C03636=1093.569,93.701,438.631,175.911,17.516,152.546
C03637=1093.575,93.950,438.614,175.913,17.517,152.546
C03638=1093.581,94.199,438.595,175.915,17.518,152.546
C03639=1093.586,94.448,438.577,175.918,17.519,152.546
C03640=1093.592,94.697,438.559,175.920,17.520,152.545
C03641=1093.598,94.947,438.541,175.923,17.521,152.545
C03642=1093.603,95.196,438.524,175.925,17.522,152.545
C03643=1093.609,95.472,438.503,175.927,17.523,152.545
C03644=1093.616,95.748,438.484,175.930,17.524,152.544
C03645=1093.622,96.023,438.464,175.933,17.525,152.544
C03646=1093.628,96.299,438.443,175.935,17.526,152.544
C03647=1093.634,96.548,438.425,175.938,17.528,152.544
C03648=1093.639,96.797,438.408,175.940,17.529,152.543
C03649=1093.645,97.048,438.389,175.942,17.530,152.543
C03650=1093.651,97.296,438.371,175.944,17.531,152.543
C03651=1093.657,97.546,438.353,175.947,17.532,152.543
C03652=1093.662,97.795,438.336,175.950,17.533,152.542
C03653=1093.668,98.045,438.317,175.952,17.534,152.542
C03654=1093.673,98.293,438.299,175.954,17.535,152.542
C03655=1093.680,98.543,438.281,175.956,17.535,152.542
C03656=1093.684,98.792,438.263,175.959,17.537,152.541
C03657=1093.691,99.041,438.244,175.961,17.537,152.541
C03658=1093.696,99.290,438.227,175.964,17.538,152.541
C03659=1093.702,99.540,438.209,175.966,17.540,152.541
C03660=1093.707,99.789,438.190,175.968,17.540,152.540
C03661=1093.714,100.039,438.172,175.971,17.541,152.540
C03662=1093.719,100.288,438.154,175.973,17.542,152.540
C03663=1093.725,100.537,438.135,175.976,17.543,152.540
C03664=1093.730,100.786,438.117,175.978,17.545,152.539
C03665=1093.736,101.036,438.099,175.980,17.545,152.539
C03666=1093.742,101.285,438.081,175.983,17.546,152.539
C03667=1093.748,101.534,438.063,175.985,17.547,152.538
C03668=1093.753,101.783,438.044,175.988,17.548,152.538
C03669=1093.759,102.033,438.026,175.990,17.549,152.538
C03670=1093.764,102.282,438.007,175.992,17.550,152.538
C03671=1093.770,102.531,437.989,175.995,17.551,152.537
C03672=1093.775,102.781,437.971,175.998,17.552,152.537
C03673=1093.781,103.030,437.952,176.000,17.553,152.537
C03674=1093.786,103.279,437.934,176.002,17.554,152.537
C03675=1093.792,103.528,437.915,176.004,17.555,152.536
C03676=1093.797,103.778,437.897,176.007,17.556,152.536
C03677=1093.804,104.027,437.879,176.010,17.557,152.536
C03678=1093.808,104.276,437.860,176.012,17.558,152.536
C03679=1093.815,104.525,437.842,176.014,17.559,152.535
C03680=1093.820,104.775,437.824,176.016,17.559,152.535
C03681=1093.826,105.024,437.805,176.019,17.560,152.535
C03682=1093.831,105.273,437.787,176.022,17.562,152.534
C03683=1093.837,105.522,437.768,176.024,17.562,152.534
C03684=1093.842,105.771,437.749,176.027,17.563,152.534
C03685=1093.848,106.021,437.731,176.029,17.565,152.534
C03686=1093.854,106.269,437.712,176.031,17.565,152.533
C03687=1093.859,106.519,437.694,176.034,17.566,152.533
C03688=1093.865,106.769,437.675,176.036,17.567,152.533
C03689=1093.870,107.017,437.656,176.039,17.568,152.532
C03690=1093.877,107.267,437.638,176.041,17.569,152.532
C03691=1093.882,107.516,437.620,176.043,17.570,152.532
C03692=1093.887,107.766,437.601,176.046,17.571,152.532
C03693=1093.893,108.015,437.582,176.049,17.572,152.531
C03694=1093.899,108.264,437.564,176.051,17.573,152.531
C03695=1093.905,108.513,437.546,176.054,17.573,152.531
C03696=1093.910,108.762,437.527,176.056,17.574,152.530
C03697=1093.915,109.012,437.508,176.058,17.575,152.530
C03698=1093.922,109.261,437.490,176.061,17.576,152.530
C03699=1093.927,109.510,437.471,176.063,17.577,152.530
C03700=1093.933,109.759,437.452,176.066,17.578,152.529
C03701=1093.939,110.009,437.433,176.069,17.579,152.529
C03702=1093.944,110.258,437.415,176.071,17.580,152.529
C03703=1093.950,110.507,437.396,176.073,17.581,152.528
C03704=1093.956,110.757,437.377,176.075,17.581,152.528
C03705=1093.962,111.005,437.358,176.078,17.582,152.528
C03706=1093.967,111.255,437.340,176.081,17.583,152.528
C03707=1093.973,111.531,437.319,176.084,17.584,152.527
C03708=1093.979,111.806,437.298,176.087,17.585,152.527
C03709=1093.985,112.082,437.277,176.089,17.586,152.527
C03710=1093.992,112.359,437.256,176.092,17.587,152.526
C03711=1093.997,112.607,437.238,176.094,17.588,152.526
C03712=1094.003,112.856,437.219,176.097,17.589,152.526
C03713=1094.009,113.106,437.199,176.099,17.589,152.525
C03714=1094.014,113.355,437.181,176.102,17.590,152.525
C03715=1094.020,113.604,437.163,176.105,17.592,152.525
C03716=1094.026,113.854,437.143,176.107,17.592,152.524
C03717=1094.031,114.103,437.124,176.109,17.593,152.524
C03718=1094.036,114.352,437.105,176.112,17.594,152.524
C03719=1094.043,114.601,437.087,176.114,17.595,152.524
C03720=1094.049,114.850,437.067,176.117,17.595,152.523
C03721=1094.054,115.099,437.048,176.120,17.597,152.523
C03722=1094.059,115.349,437.029,176.122,17.597,152.523
C03723=1094.065,115.598,437.010,176.124,17.598,152.522
C03724=1094.070,115.847,436.991,176.127,17.599,152.522
C03725=1094.076,116.096,436.972,176.129,17.600,152.522
C03726=1094.081,116.346,436.953,176.132,17.601,152.521
C03727=1094.086,116.595,436.934,176.134,17.602,152.521
C03728=1094.092,116.844,436.915,176.137,17.602,152.521
C03729=1094.098,117.094,436.896,176.140,17.604,152.520
C03730=1094.103,117.343,436.877,176.142,17.604,152.520
C03731=1094.108,117.592,436.858,176.145,17.605,152.520
C03732=1094.114,117.842,436.839,176.147,17.606,152.520
C03733=1094.119,118.090,436.820,176.149,17.607,152.519
C03734=1094.126,118.339,436.801,176.152,17.607,152.519
C03735=1094.132,118.588,436.781,176.155,17.609,152.519
C03736=1094.137,118.838,436.762,176.157,17.609,152.518
C03737=1094.142,119.086,436.743,176.160,17.610,152.518
C03738=1094.148,119.336,436.724,176.163,17.611,152.518
C03739=1094.154,119.585,436.705,176.165,17.611,152.517
C03740=1094.159,119.835,436.685,176.167,17.613,152.517
C03741=1094.165,120.083,436.666,176.170,17.614,152.517
C03742=1094.170,120.333,436.647,176.172,17.614,152.516
C03743=1094.176,120.582,436.628,176.175,17.615,152.516
C03744=1094.182,120.832,436.609,176.178,17.616,152.516
C03745=1094.187,121.080,436.590,176.181,17.617,152.515
C03746=1094.193,121.329,436.570,176.183,17.617,152.515
C03747=1094.198,121.579,436.551,176.186,17.618,152.515
C03748=1094.204,121.828,436.531,176.188,17.620,152.515
C03749=1094.210,122.078,436.512,176.191,17.620,152.514
C03750=1094.215,122.326,436.493,176.193,17.621,152.514
C03751=1094.220,122.575,436.473,176.196,17.622,152.513
C03752=1094.226,122.825,436.453,176.198,17.622,152.513
C03753=1094.231,123.074,436.434,176.201,17.623,152.513
C03754=1094.237,123.324,436.415,176.204,17.624,152.512
C03755=1094.242,123.572,436.396,176.206,17.624,152.512
C03756=1094.248,123.821,436.376,176.209,17.626,152.512
C03757=1094.254,124.071,436.357,176.212,17.626,152.511
C03758=1094.260,124.320,436.338,176.214,17.627,152.511
C03759=1094.266,124.569,436.318,176.217,17.628,152.511
C03760=1094.271,124.818,436.298,176.220,17.628,152.510
C03761=1094.277,125.068,436.279,176.222,17.629,152.510
C03762=1094.282,125.316,436.260,176.225,17.630,152.510
C03763=1094.288,125.565,436.240,176.227,17.631,152.509
C03764=1094.294,125.815,436.221,176.229,17.631,152.509
C03765=1094.299,126.064,436.202,176.232,17.632,152.509
C03766=1094.305,126.313,436.181,176.235,17.633,152.508
C03767=1094.310,126.563,436.162,176.238,17.634,152.508
C03768=1094.316,126.812,436.142,176.240,17.634,152.508
C03769=1094.322,127.061,436.123,176.243,17.635,152.507
C03770=1094.328,127.310,436.104,176.246,17.636,152.507
C03771=1094.334,127.586,436.082,176.249,17.637,152.506
C03772=1094.340,127.862,436.060,176.252,17.638,152.506
C03773=1094.347,128.138,436.039,176.255,17.639,152.506
C03774=1094.353,128.413,436.017,176.258,17.639,152.505
C03775=1094.358,128.663,435.997,176.260,17.639,152.505
C03776=1094.364,128.912,435.977,176.263,17.641,152.505
C03777=1094.370,129.161,435.958,176.266,17.641,152.504
C03778=1094.376,129.410,435.938,176.268,17.642,152.504
C03779=1094.382,129.659,435.919,176.271,17.642,152.503
C03780=1094.388,129.908,435.899,176.274,17.643,152.503
C03781=1094.393,130.158,435.879,176.276,17.644,152.503
C03782=1094.398,130.407,435.859,176.279,17.644,152.502
C03783=1094.404,130.656,435.840,176.282,17.645,152.502
C03784=1094.410,130.905,435.820,176.284,17.646,152.502
C03785=1094.416,131.154,435.800,176.287,17.646,152.501
C03786=1094.422,131.403,435.780,176.290,17.647,152.501
C03787=1094.427,131.653,435.761,176.293,17.648,152.500
C03788=1094.433,131.902,435.741,176.294,17.649,152.500
C03789=1094.439,132.151,435.721,176.297,17.649,152.500
C03790=1094.444,132.400,435.701,176.300,17.650,152.499
C03791=1094.450,132.649,435.681,176.303,17.650,152.499
C03792=1094.455,132.898,435.662,176.305,17.651,152.499
C03793=1094.461,133.147,435.642,176.308,17.652,152.498
C03794=1094.466,133.396,435.621,176.311,17.653,152.498
C03795=1094.472,133.645,435.602,176.313,17.653,152.498
C03796=1094.477,133.894,435.582,176.316,17.654,152.497
C03797=1094.483,134.144,435.562,176.319,17.655,152.497
C03798=1094.489,134.393,435.542,176.322,17.656,152.496
C03799=1094.494,134.642,435.522,176.324,17.656,152.496
C03800=1094.500,134.891,435.502,176.327,17.657,152.496
C03801=1094.505,135.140,435.482,176.330,17.658,152.495
C03802=1094.511,135.389,435.462,176.332,17.658,152.495
C03803=1094.517,135.638,435.442,176.335,17.659,152.495
C03804=1094.522,135.888,435.422,176.338,17.659,152.494
C03805=1094.528,136.137,435.402,176.341,17.661,152.494
C03806=1094.534,136.386,435.381,176.343,17.661,152.493
C03807=1094.540,136.635,435.362,176.346,17.661,152.493
C03808=1094.545,136.885,435.342,176.349,17.662,152.493
C03809=1094.551,137.134,435.322,176.352,17.663,152.492
C03810=1094.557,137.383,435.302,176.354,17.663,152.492
C03811=1094.562,137.632,435.281,176.357,17.664,152.492
C03812=1094.568,137.880,435.261,176.360,17.665,152.491
C03813=1094.573,138.130,435.241,176.362,17.665,152.491
C03814=1094.579,138.379,435.221,176.365,17.666,152.490
C03815=1094.584,138.628,435.201,176.368,17.667,152.490
C03816=1094.590,138.877,435.181,176.371,17.667,152.490
C03817=1094.595,139.126,435.160,176.373,17.668,152.489
C03818=1094.601,139.375,435.140,176.376,17.668,152.489
C03819=1094.606,139.625,435.121,176.379,17.669,152.488
C03820=1094.613,139.874,435.100,176.382,17.670,152.488
C03821=1094.618,140.123,435.080,176.384,17.670,152.488
C03822=1094.624,140.372,435.060,176.387,17.671,152.487
C03823=1094.629,140.621,435.039,176.390,17.672,152.487
C03824=1094.635,140.870,435.019,176.393,17.673,152.486
C03825=1094.641,141.119,434.999,176.395,17.673,152.486
C03826=1094.646,141.368,434.978,176.398,17.674,152.486
C03827=1094.652,141.617,434.958,176.401,17.674,152.485
C03828=1094.657,141.866,434.938,176.404,17.675,152.485
C03829=1094.662,142.115,434.917,176.406,17.675,152.484
C03830=1094.669,142.365,434.897,176.409,17.676,152.484
C03831=1094.674,142.614,434.876,176.412,17.677,152.484
C03832=1094.679,142.863,434.856,176.415,17.677,152.483
C03833=1094.685,143.112,434.836,176.418,17.678,152.483
C03834=1094.691,143.361,434.815,176.420,17.679,152.482
C03835=1094.697,143.637,434.793,176.424,17.679,152.482
C03836=1094.703,143.913,434.770,176.427,17.680,152.482
C03837=1094.709,144.189,434.747,176.430,17.681,152.481
C03838=1094.715,144.464,434.725,176.432,17.681,152.481
C03839=1094.721,144.713,434.705,176.435,17.682,152.480
C03840=1094.726,144.962,434.684,176.438,17.683,152.480
C03841=1094.732,145.212,434.663,176.441,17.683,152.479
C03842=1094.739,145.460,434.643,176.444,17.684,152.479
C03843=1094.744,145.709,434.622,176.447,17.684,152.479
C03844=1094.749,145.958,434.601,176.450,17.685,152.478
C03845=1094.754,146.208,434.581,176.453,17.685,152.478
C03846=1094.761,146.457,434.561,176.455,17.686,152.477
C03847=1094.766,146.706,434.540,176.458,17.686,152.477
C03848=1094.771,146.955,434.519,176.461,17.687,152.476
C03849=1094.778,147.203,434.499,176.464,17.688,152.476
C03850=1094.784,147.453,434.478,176.467,17.689,152.476
C03851=1094.789,147.702,434.457,176.469,17.689,152.475
C03852=1094.794,147.952,434.437,176.472,17.689,152.475
C03853=1094.800,148.200,434.417,176.475,17.690,152.474
C03854=1094.806,148.449,434.396,176.478,17.690,152.474
C03855=1094.812,148.699,434.375,176.481,17.691,152.473
C03856=1094.817,148.948,434.354,176.484,17.691,152.473
C03857=1094.822,149.197,434.334,176.487,17.692,152.473
C03858=1094.828,149.445,434.312,176.490,17.693,152.472
C03859=1094.834,149.695,434.292,176.493,17.694,152.472
C03860=1094.839,149.944,434.271,176.495,17.694,152.471
C03861=1094.845,150.193,434.250,176.498,17.694,152.471
C03862=1094.850,150.442,434.230,176.501,17.695,152.471
C03863=1094.856,150.692,434.209,176.504,17.695,152.470
C03864=1094.862,150.940,434.187,176.506,17.696,152.470
C03865=1094.867,151.189,434.167,176.509,17.696,152.469
C03866=1094.872,151.438,434.146,176.512,17.697,152.469
C03867=1094.878,151.687,434.125,176.515,17.698,152.468
C03868=1094.884,151.936,434.105,176.518,17.699,152.468
C03869=1094.890,152.185,434.084,176.520,17.698,152.467
C03870=1094.896,152.435,434.062,176.523,17.699,152.467
C03871=1094.901,152.684,434.042,176.526,17.700,152.467
C03872=1094.907,152.932,434.021,176.529,17.701,152.466
C03873=1094.912,153.181,434.000,176.532,17.701,152.466
C03874=1094.918,153.431,433.979,176.535,17.701,152.465
C03875=1094.923,153.680,433.958,176.538,17.702,152.465
C03876=1094.929,153.929,433.937,176.541,17.702,152.464
C03877=1094.935,154.178,433.916,176.544,17.703,152.464
C03878=1094.940,154.427,433.895,176.547,17.704,152.463
C03879=1094.946,154.676,433.874,176.549,17.704,152.463
C03880=1094.951,154.925,433.853,176.552,17.704,152.463
C03881=1094.957,155.174,433.832,176.555,17.705,152.462
C03882=1094.962,155.423,433.811,176.559,17.705,152.462
C03883=1094.968,155.672,433.790,176.561,17.706,152.461
C03884=1094.974,155.921,433.769,176.564,17.706,152.461
C03885=1094.979,156.170,433.748,176.567,17.707,152.460
C03886=1094.985,156.420,433.727,176.570,17.707,152.460
C03887=1094.991,156.668,433.706,176.573,17.708,152.460
C03888=1094.997,156.917,433.684,176.576,17.709,152.459
C03889=1095.002,157.167,433.663,176.578,17.709,152.459
C03890=1095.008,157.415,433.642,176.581,17.709,152.458
C03891=1095.013,157.665,433.621,176.584,17.710,152.458
C03892=1095.018,157.914,433.599,176.587,17.711,152.457
C03893=1095.024,158.162,433.578,176.591,17.711,152.457
C03894=1095.030,158.412,433.557,176.594,17.712,152.456
C03895=1095.035,158.661,433.536,176.596,17.712,152.456
C03896=1095.041,158.910,433.514,176.599,17.712,152.455
C03897=1095.047,159.159,433.494,176.602,17.713,152.455
C03898=1095.052,159.407,433.472,176.605,17.714,152.455
C03899=1095.058,159.683,433.448,176.608,17.714,152.454
C03900=1095.065,159.958,433.425,176.611,17.714,152.453
C03901=1095.071,160.234,433.401,176.614,17.715,152.453
C03902=1095.077,160.509,433.378,176.618,17.715,152.453
C03903=1095.083,160.759,433.357,176.621,17.716,152.452
C03904=1095.088,161.008,433.335,176.624,17.716,152.452
C03905=1095.094,161.256,433.314,176.627,17.717,152.451
C03906=1095.099,161.506,433.292,176.630,17.717,152.451
C03907=1095.105,161.754,433.271,176.632,17.718,152.450
C03908=1095.111,162.004,433.250,176.635,17.718,152.450
C03909=1095.116,162.253,433.228,176.639,17.719,152.449
C03910=1095.121,162.501,433.207,176.642,17.719,152.449
C03911=1095.127,162.751,433.185,176.645,17.720,152.448
C03912=1095.132,162.999,433.163,176.648,17.720,152.448
C03913=1095.138,163.249,433.142,176.651,17.721,152.447
C03914=1095.143,163.498,433.120,176.653,17.721,152.447
C03915=1095.149,163.747,433.099,176.656,17.722,152.446
C03916=1095.155,163.996,433.077,176.659,17.722,152.446
C03917=1095.159,164.245,433.055,176.662,17.723,152.446
C03918=1095.166,164.494,433.034,176.665,17.723,152.445
C03919=1095.170,164.743,433.012,176.668,17.724,152.445
C03920=1095.176,164.992,432.991,176.671,17.724,152.444
C03921=1095.181,165.241,432.969,176.674,17.725,152.444
C03922=1095.187,165.490,432.948,176.677,17.725,152.443
C03923=1095.193,165.739,432.926,176.680,17.726,152.443
C03924=1095.198,165.988,432.904,176.683,17.726,152.442
C03925=1095.204,166.237,432.883,176.686,17.727,152.442
C03926=1095.209,166.486,432.861,176.689,17.728,152.441
C03927=1095.215,166.735,432.839,176.691,17.728,152.441
C03928=1095.220,166.984,432.817,176.695,17.728,152.440
C03929=1095.226,167.233,432.796,176.698,17.729,152.440
C03930=1095.231,167.482,432.774,176.701,17.729,152.439
C03931=1095.237,167.731,432.752,176.704,17.730,152.439
C03932=1095.242,167.980,432.730,176.707,17.730,152.439
C03933=1095.248,168.229,432.709,176.710,17.731,152.438
C03934=1095.253,168.478,432.687,176.713,17.731,152.438
C03935=1095.259,168.727,432.665,176.716,17.731,152.437
C03936=1095.264,168.975,432.643,176.719,17.732,152.437
C03937=1095.270,169.224,432.621,176.722,17.732,152.436
C03938=1095.276,169.474,432.599,176.725,17.733,152.436
C03939=1095.281,169.723,432.578,176.728,17.733,152.435
C03940=1095.287,169.972,432.555,176.731,17.734,152.435
C03941=1095.292,170.221,432.534,176.734,17.734,152.434
C03942=1095.297,170.470,432.512,176.737,17.734,152.434
C03943=1095.303,170.719,432.491,176.740,17.735,152.433
C03944=1095.309,170.967,432.468,176.743,17.735,152.433
C03945=1095.315,171.217,432.446,176.746,17.735,152.432
C03946=1095.320,171.465,432.424,176.749,17.736,152.432
C03947=1095.326,171.715,432.402,176.752,17.737,152.431
C03948=1095.331,171.963,432.381,176.755,17.737,152.431
C03949=1095.336,172.212,432.358,176.759,17.738,152.430
C03950=1095.343,172.462,432.336,176.761,17.737,152.430
C03951=1095.347,172.710,432.314,176.764,17.738,152.429
C03952=1095.354,172.960,432.293,176.767,17.738,152.429
C03953=1095.359,173.208,432.270,176.770,17.739,152.428
C03954=1095.365,173.457,432.248,176.774,17.739,152.428
C03955=1095.370,173.707,432.226,176.777,17.740,152.427
C03956=1095.375,173.955,432.204,176.780,17.740,152.427
C03957=1095.382,174.204,432.182,176.783,17.741,152.426
C03958=1095.387,174.453,432.160,176.786,17.740,152.426
C03959=1095.393,174.702,432.138,176.789,17.741,152.425
C03960=1095.398,174.951,432.115,176.792,17.742,152.425
C03961=1095.404,175.200,432.093,176.795,17.742,152.424
C03962=1095.410,175.448,432.071,176.798,17.742,152.424
C03963=1095.416,175.724,432.047,176.802,17.742,152.423
C03964=1095.422,175.999,432.022,176.805,17.743,152.423
C03965=1095.428,176.274,431.998,176.809,17.744,152.422
C03966=1095.434,176.549,431.973,176.812,17.744,152.421
C03967=1095.440,176.798,431.951,176.815,17.745,152.421
C03968=1095.446,177.047,431.928,176.818,17.745,152.420
C03969=1095.451,177.297,431.906,176.822,17.745,152.420
C03970=1095.457,177.544,431.884,176.824,17.745,152.419
C03971=1095.463,177.794,431.862,176.827,17.745,152.419
C03972=1095.468,178.043,431.839,176.830,17.746,152.418
C03973=1095.474,178.292,431.817,176.834,17.746,152.418
C03974=1095.480,178.540,431.795,176.837,17.747,152.417
C03975=1095.485,178.790,431.773,176.840,17.747,152.417
C03976=1095.491,179.038,431.750,176.843,17.747,152.416
C03977=1095.497,179.288,431.728,176.846,17.748,152.416
C03978=1095.503,179.537,431.705,176.850,17.748,152.415
C03979=1095.508,179.785,431.684,176.853,17.749,152.415
C03980=1095.514,180.034,431.661,176.855,17.748,152.414
C03981=1095.520,180.283,431.638,176.858,17.749,152.414
C03982=1095.525,180.533,431.616,176.862,17.749,152.413
C03983=1095.532,180.781,431.593,176.865,17.749,152.412
C03984=1095.536,181.030,431.571,176.868,17.750,152.412
C03985=1095.542,181.279,431.549,176.871,17.750,152.412
C03986=1095.548,181.528,431.526,176.874,17.751,152.411
C03987=1095.554,181.777,431.504,176.878,17.751,152.410
C03988=1095.560,182.026,431.481,176.881,17.751,152.410
C03989=1095.565,182.275,431.458,176.884,17.751,152.409
C03990=1095.570,182.524,431.436,176.887,17.752,152.409
C03991=1095.577,182.772,431.414,176.891,17.752,152.408
C03992=1095.582,183.021,431.391,176.893,17.752,152.408
C03993=1095.588,183.271,431.369,176.896,17.752,152.407
C03994=1095.594,183.520,431.346,176.900,17.752,152.407
C03995=1095.600,183.768,431.323,176.903,17.753,152.406
C03996=1095.606,184.017,431.300,176.906,17.753,152.405
C03997=1095.611,184.267,431.278,176.909,17.753,152.405
C03998=1095.617,184.515,431.255,176.913,17.754,152.404
C03999=1095.622,184.764,431.233,176.916,17.754,152.404
C04000=1095.629,185.012,431.210,176.919,17.754,152.403
C04001=1095.634,185.261,431.187,176.922,17.755,152.403
C04002=1095.640,185.511,431.165,176.925,17.755,152.402
C04003=1095.645,185.760,431.142,176.929,17.756,152.402
C04004=1095.650,186.009,431.119,176.932,17.756,152.401
C04005=1095.656,186.257,431.096,176.935,17.756,152.401
C04006=1095.661,186.506,431.073,176.938,17.757,152.400
C04007=1095.667,186.755,431.050,176.941,17.757,152.400
C04008=1095.672,187.004,431.028,176.944,17.757,152.399
C04009=1095.678,187.253,431.005,176.947,17.757,152.399
C04010=1095.684,187.502,430.982,176.950,17.758,152.398
C04011=1095.689,187.750,430.960,176.954,17.758,152.397
C04012=1095.694,187.999,430.936,176.957,17.758,152.397
C04013=1095.700,188.248,430.913,176.960,17.759,152.396
C04014=1095.706,188.497,430.890,176.963,17.759,152.396
C04015=1095.711,188.746,430.867,176.966,17.760,152.395
C04016=1095.717,188.995,430.844,176.970,17.760,152.395
C04017=1095.723,189.244,430.821,176.973,17.760,152.394
C04018=1095.728,189.492,430.799,176.976,17.761,152.394
C04019=1095.733,189.741,430.775,176.979,17.761,152.393
C04020=1095.739,189.990,430.752,176.983,17.761,152.393
C04021=1095.744,190.239,430.729,176.986,17.762,152.392
C04022=1095.750,190.488,430.706,176.989,17.762,152.392
C04023=1095.756,190.737,430.683,176.992,17.762,152.391
C04024=1095.761,190.986,430.660,176.996,17.763,152.390
C04025=1095.766,191.235,430.637,176.999,17.763,152.390
C04026=1095.772,191.484,430.614,177.002,17.763,152.389
C04027=1095.778,191.758,430.589,177.005,17.763,152.389
C04028=1095.784,192.034,430.563,177.009,17.764,152.388
C04029=1095.791,192.308,430.538,177.013,17.765,152.388
C04030=1095.796,192.583,430.512,177.016,17.765,152.387
C04031=1095.802,192.832,430.489,177.019,17.765,152.386
C04032=1095.808,193.081,430.466,177.023,17.765,152.386
C04033=1095.813,193.329,430.443,177.026,17.765,152.385
C04034=1095.819,193.578,430.419,177.029,17.766,152.385
C04035=1095.824,193.827,430.396,177.032,17.766,152.384
C04036=1095.830,194.076,430.373,177.036,17.766,152.384
C04037=1095.836,194.325,430.350,177.039,17.767,152.383
C04038=1095.842,194.574,430.327,177.042,17.767,152.382
C04039=1095.847,194.822,430.303,177.045,17.767,152.382
C04040=1095.853,195.071,430.280,177.049,17.768,152.381
C04041=1095.858,195.320,430.257,177.052,17.768,152.381
C04042=1095.863,195.569,430.233,177.055,17.768,152.380
C04043=1095.869,195.818,430.209,177.058,17.769,152.380
C04044=1095.875,196.066,430.187,177.062,17.769,152.379
C04045=1095.881,196.315,430.164,177.065,17.769,152.378
C04046=1095.886,196.564,430.139,177.068,17.769,152.378
C04047=1095.892,196.813,430.116,177.072,17.769,152.377
C04048=1095.898,197.062,430.093,177.075,17.770,152.377
C04049=1095.904,197.311,430.069,177.078,17.770,152.376
C04050=1095.909,197.560,430.046,177.081,17.770,152.376
C04051=1095.915,197.809,430.023,177.085,17.771,152.375
C04052=1095.920,198.057,429.999,177.088,17.771,152.375
C04053=1095.926,198.306,429.976,177.091,17.771,152.374
C04054=1095.932,198.555,429.953,177.095,17.771,152.373
C04055=1095.937,198.804,429.928,177.098,17.772,152.373
C04056=1095.943,199.053,429.906,177.101,17.772,152.372
C04057=1095.949,199.301,429.882,177.104,17.772,152.372
C04058=1095.954,199.550,429.858,177.108,17.772,152.371
C04059=1095.960,199.799,429.834,177.111,17.772,152.370
C04060=1095.965,200.048,429.811,177.114,17.773,152.370
C04061=1095.972,200.297,429.787,177.118,17.773,152.369
C04062=1095.977,200.545,429.764,177.121,17.773,152.369
C04063=1095.983,200.794,429.740,177.124,17.773,152.368
C04064=1095.988,201.043,429.717,177.128,17.774,152.368
C04065=1095.995,201.292,429.693,177.131,17.774,152.367
C04066=1096.000,201.541,429.669,177.134,17.774,152.366
C04067=1096.006,201.789,429.646,177.138,17.774,152.366
C04068=1096.011,202.039,429.622,177.141,17.774,152.365
C04069=1096.017,202.287,429.599,177.144,17.775,152.365
C04070=1096.023,202.537,429.575,177.147,17.775,152.364
C04071=1096.029,202.785,429.551,177.151,17.775,152.363
C04072=1096.034,203.034,429.527,177.154,17.775,152.363
C04073=1096.040,203.283,429.504,177.157,17.776,152.362
C04074=1096.045,203.531,429.480,177.161,17.776,152.362
C04075=1096.051,203.780,429.457,177.164,17.776,152.361
C04076=1096.057,204.029,429.432,177.167,17.777,152.361
C04077=1096.063,204.278,429.408,177.171,17.776,152.360
C04078=1096.068,204.527,429.385,177.174,17.777,152.359
C04079=1096.073,204.775,429.360,177.177,17.777,152.359
C04080=1096.079,205.024,429.337,177.180,17.777,152.358
C04081=1096.084,205.273,429.313,177.184,17.778,152.358
C04082=1096.090,205.522,429.289,177.187,17.778,152.357
C04083=1096.096,205.770,429.265,177.190,17.778,152.357
C04084=1096.101,206.019,429.241,177.194,17.778,152.356
C04085=1096.106,206.268,429.217,177.197,17.779,152.355
C04086=1096.112,206.517,429.194,177.200,17.779,152.355
C04087=1096.118,206.766,429.169,177.204,17.779,152.354
C04088=1096.123,207.014,429.145,177.207,17.779,152.354
C04089=1096.129,207.263,429.121,177.211,17.780,152.353
C04090=1096.134,207.512,429.097,177.214,17.780,152.353
C04091=1096.158,208.525,428.999,177.264,17.800,152.347
C04092=1096.166,208.898,428.963,177.269,17.802,152.347
C04093=1096.175,209.271,428.927,177.274,17.804,152.346
C04094=1096.183,209.644,428.889,177.279,17.805,152.346
C04095=1096.192,210.017,428.853,177.283,17.807,152.345
C04096=1096.197,210.265,428.828,177.286,17.808,152.345
C04097=1096.202,210.514,428.804,177.290,17.809,152.344
C04098=1096.208,210.763,428.780,177.293,17.810,152.344
C04099=1096.214,211.012,428.755,177.296,17.811,152.344
C04100=1096.220,211.260,428.732,177.300,17.813,152.343
C04101=1096.226,211.509,428.707,177.302,17.814,152.343
C04102=1096.231,211.758,428.683,177.305,17.814,152.343
C04103=1096.237,212.007,428.658,177.309,17.816,152.342
C04104=1096.242,212.255,428.633,177.312,17.817,152.342
C04105=1096.248,212.504,428.609,177.316,17.818,152.341
C04106=1096.254,212.753,428.584,177.319,17.819,152.341
C04107=1096.259,213.002,428.560,177.321,17.821,152.341
C04108=1096.265,213.251,428.535,177.325,17.822,152.340
C04109=1096.270,213.499,428.510,177.328,17.823,152.340
C04110=1096.276,213.748,428.486,177.331,17.824,152.340
C04111=1096.282,213.997,428.462,177.335,17.825,152.339
C04112=1096.287,214.245,428.437,177.338,17.826,152.339
C04113=1096.292,214.494,428.411,177.341,17.827,152.339
C04114=1096.298,214.743,428.387,177.344,17.829,152.338
C04115=1096.304,214.992,428.363,177.347,17.830,152.338
C04116=1096.309,215.240,428.338,177.351,17.831,152.338
C04117=1096.314,215.489,428.313,177.354,17.832,152.337
C04118=1096.320,215.738,428.289,177.356,17.833,152.337
C04119=1096.326,215.986,428.264,177.360,17.834,152.337
C04120=1096.332,216.235,428.239,177.363,17.836,152.336
C04121=1096.337,216.484,428.214,177.366,17.836,152.336
C04122=1096.343,216.733,428.189,177.370,17.838,152.335
C04123=1096.348,216.982,428.165,177.373,17.839,152.335
C04124=1096.354,217.230,428.139,177.376,17.841,152.335
C04125=1096.359,217.479,428.115,177.379,17.841,152.334
C04126=1096.366,217.727,428.090,177.382,17.842,152.334
C04127=1096.371,217.976,428.065,177.386,17.844,152.334
C04128=1096.376,218.225,428.040,177.389,17.845,152.333
C04129=1096.382,218.474,428.015,177.392,17.846,152.333
C04130=1096.388,218.722,427.990,177.395,17.847,152.333
C04131=1096.393,218.971,427.966,177.398,17.848,152.332
C04132=1096.399,219.220,427.940,177.402,17.850,152.332
C04133=1096.404,219.468,427.915,177.405,17.850,152.332
C04134=1096.410,219.717,427.890,177.409,17.852,152.331
C04135=1096.415,219.966,427.866,177.411,17.853,152.331
C04136=1096.422,220.214,427.841,177.414,17.854,152.331
C04137=1096.427,220.464,427.815,177.418,17.855,152.330
C04138=1096.432,220.712,427.790,177.421,17.857,152.330
C04139=1096.439,220.961,427.765,177.425,17.858,152.329
C04140=1096.444,221.209,427.741,177.427,17.859,152.329
C04141=1096.450,221.458,427.715,177.430,17.860,152.329
C04142=1096.455,221.707,427.690,177.434,17.861,152.328
C04143=1096.461,221.955,427.665,177.437,17.862,152.328
C04144=1096.470,222.332,427.627,177.442,17.864,152.327
C04145=1096.478,222.709,427.589,177.447,17.866,152.327
C04146=1096.487,223.086,427.550,177.452,17.868,152.326
C04147=1096.495,223.463,427.512,177.457,17.870,152.326
C04148=1096.500,223.711,427.487,177.460,17.870,152.326
C04149=1096.506,223.959,427.462,177.463,17.872,152.325
C04150=1096.512,224.208,427.436,177.466,17.873,152.325
C04151=1096.517,224.457,427.412,177.470,17.875,152.324
C04152=1096.523,224.706,427.386,177.473,17.876,152.324
C04153=1096.529,224.954,427.361,177.476,17.877,152.324
C04154=1096.534,225.203,427.335,177.479,17.878,152.323
C04155=1096.540,225.451,427.310,177.483,17.880,152.323
C04156=1096.545,225.701,427.284,177.486,17.881,152.323
C04157=1096.551,225.949,427.259,177.489,17.881,152.322
C04158=1096.556,226.198,427.234,177.493,17.883,152.322
C04159=1096.562,226.446,427.209,177.495,17.884,152.322
C04160=1096.568,226.695,427.183,177.499,17.886,152.321
C04161=1096.573,226.944,427.157,177.502,17.886,152.321
C04162=1096.580,227.192,427.132,177.505,17.888,152.321
C04163=1096.584,227.441,427.106,177.508,17.889,152.320
C04164=1096.591,227.689,427.081,177.512,17.890,152.320
C04165=1096.596,227.938,427.055,177.515,17.892,152.320
C04166=1096.601,228.186,427.030,177.518,17.892,152.319
C04167=1096.607,228.435,427.004,177.522,17.894,152.319
C04168=1096.613,228.684,426.978,177.524,17.895,152.319
C04169=1096.619,228.933,426.953,177.528,17.897,152.318
C04170=1096.624,229.181,426.927,177.531,17.897,152.318
C04171=1096.630,229.430,426.902,177.535,17.899,152.318
C04172=1096.635,229.679,426.876,177.538,17.900,152.317
C04173=1096.642,229.927,426.851,177.541,17.901,152.317
C04174=1096.647,230.176,426.825,177.544,17.903,152.317
C04175=1096.653,230.424,426.800,177.548,17.904,152.316
C04176=1096.658,230.673,426.774,177.551,17.905,152.316
C04177=1096.664,230.922,426.748,177.554,17.907,152.316
C04178=1096.669,231.170,426.723,177.557,17.908,152.315
C04179=1096.675,231.419,426.697,177.561,17.909,152.315
C04180=1096.680,231.668,426.671,177.564,17.910,152.315
C04181=1096.686,231.917,426.644,177.568,17.912,152.314
C04182=1096.692,232.165,426.620,177.570,17.913,152.314
C04183=1096.697,232.414,426.594,177.573,17.914,152.314
C04184=1096.703,232.663,426.568,177.577,17.915,152.313
C04185=1096.709,232.911,426.542,177.580,17.916,152.313
C04186=1096.715,233.160,426.516,177.583,17.918,152.312
C04187=1096.719,233.408,426.490,177.586,17.919,152.312
C04188=1096.725,233.657,426.464,177.590,17.920,152.312
C04189=1096.731,233.905,426.439,177.593,17.921,152.311
C04190=1096.737,234.154,426.412,177.596,17.923,152.311
C04191=1096.742,234.403,426.386,177.599,17.924,152.311
C04192=1096.748,234.652,426.360,177.603,17.925,152.310
C04193=1096.753,234.900,426.335,177.606,17.927,152.310
C04194=1096.759,235.148,426.309,177.610,17.928,152.310
C04195=1096.765,235.397,426.283,177.612,17.929,152.310
C04196=1096.773,235.765,426.244,177.618,17.931,152.309
C04197=1096.781,236.133,426.206,177.623,17.933,152.309
C04198=1096.790,236.501,426.167,177.627,17.935,152.308
C04199=1096.798,236.869,426.128,177.632,17.937,152.308
C04200=1096.803,237.118,426.103,177.635,17.939,152.307
C04201=1096.809,237.366,426.076,177.638,17.940,152.307
C04202=1096.814,237.615,426.050,177.642,17.941,152.307
C04203=1096.820,237.864,426.023,177.645,17.942,152.306
C04204=1096.826,238.113,425.997,177.649,17.944,152.306
C04205=1096.831,238.361,425.971,177.651,17.945,152.306
C04206=1096.837,238.610,425.945,177.655,17.946,152.305
C04207=1096.843,238.858,425.918,177.658,17.948,152.305
C04208=1096.848,239.107,425.892,177.662,17.949,152.305
C04209=1096.854,239.356,425.866,177.664,17.950,152.304
C04210=1096.860,239.604,425.841,177.668,17.952,152.304
C04211=1096.865,239.852,425.814,177.672,17.953,152.304
C04212=1096.871,240.101,425.788,177.675,17.954,152.303
C04213=1096.877,240.349,425.761,177.678,17.956,152.303
C04214=1096.882,240.598,425.735,177.681,17.957,152.303
C04215=1096.888,240.847,425.709,177.685,17.958,152.302
C04216=1096.894,241.095,425.682,177.688,17.959,152.302
C04217=1096.899,241.344,425.656,177.691,17.961,152.302
C04218=1096.905,241.592,425.630,177.694,17.962,152.301
C04219=1096.911,241.841,425.603,177.698,17.964,152.301
C04220=1096.916,242.090,425.577,177.701,17.965,152.301
C04221=1096.922,242.338,425.550,177.704,17.966,152.300
C04222=1096.928,242.586,425.524,177.707,17.967,152.300
C04223=1096.933,242.835,425.497,177.711,17.969,152.300
C04224=1096.939,243.084,425.471,177.714,17.971,152.299
C04225=1096.944,243.332,425.444,177.717,17.971,152.299
C04226=1096.950,243.581,425.417,177.721,17.973,152.299
C04227=1096.955,243.829,425.391,177.724,17.974,152.298
C04228=1096.961,244.078,425.365,177.727,17.976,152.298
C04229=1096.967,244.326,425.338,177.730,17.977,152.298
C04230=1096.972,244.575,425.311,177.734,17.979,152.298
C04231=1096.977,244.824,425.284,177.738,17.980,152.297
C04232=1096.983,245.072,425.257,177.740,17.981,152.297
C04233=1096.989,245.321,425.232,177.744,17.983,152.296
C04234=1096.994,245.569,425.205,177.747,17.984,152.296
C04235=1097.000,245.818,425.178,177.750,17.986,152.296
C04236=1097.005,246.066,425.151,177.753,17.987,152.296
C04237=1097.011,246.315,425.124,177.757,17.988,152.295
C04238=1097.017,246.563,425.098,177.761,17.990,152.295
C04239=1097.023,246.811,425.071,177.763,17.991,152.295
C04240=1097.028,247.060,425.044,177.767,17.993,152.294
C04241=1097.034,247.309,425.017,177.770,17.994,152.294
C04242=1097.040,247.557,424.990,177.773,17.995,152.294
C04243=1097.046,247.806,424.963,177.776,17.997,152.294
C04244=1097.051,248.054,424.936,177.780,17.998,152.293
C04245=1097.056,248.303,424.910,177.783,18.000,152.293
C04246=1097.061,248.551,424.882,177.786,18.001,152.293
C04247=1097.067,248.800,424.856,177.790,18.003,152.292
C04248=1097.075,249.161,424.817,177.794,18.005,152.292
C04249=1097.083,249.522,424.778,177.799,18.006,152.291
C04250=1097.091,249.884,424.739,177.804,18.009,152.291
C04251=1097.099,250.245,424.699,177.809,18.011,152.291
C04252=1097.105,250.493,424.672,177.812,18.012,152.290
C04253=1097.110,250.742,424.645,177.815,18.014,152.290
C04254=1097.116,250.990,424.619,177.819,18.016,152.290
C04255=1097.122,251.238,424.591,177.822,18.017,152.289
C04256=1097.127,251.487,424.564,177.825,18.018,152.289
C04257=1097.133,251.736,424.537,177.829,18.020,152.289
C04258=1097.138,251.985,424.510,177.832,18.021,152.289
C04259=1097.144,252.233,424.483,177.835,18.023,152.288
C04260=1097.149,252.481,424.455,177.838,18.024,152.288
C04261=1097.155,252.729,424.428,177.842,18.026,152.288
C04262=1097.160,252.978,424.401,177.845,18.027,152.287
C04263=1097.166,253.227,424.374,177.848,18.029,152.287
C04264=1097.172,253.475,424.346,177.852,18.030,152.287
C04265=1097.177,253.723,424.320,177.855,18.031,152.287
C04266=1097.182,253.972,424.292,177.858,18.033,152.286
C04267=1097.189,254.220,424.265,177.862,18.035,152.286
C04268=1097.194,254.469,424.237,177.865,18.036,152.286
C04269=1097.200,254.718,424.211,177.868,18.037,152.285
C04270=1097.205,254.966,424.183,177.872,18.039,152.285
C04271=1097.211,255.214,424.156,177.874,18.041,152.285
C04272=1097.217,255.463,424.128,177.878,18.042,152.284
C04273=1097.222,255.711,424.101,177.882,18.044,152.284
C04274=1097.228,255.960,424.074,177.885,18.045,152.284
C04275=1097.233,256.208,424.046,177.888,18.046,152.284
C04276=1097.240,256.457,424.019,177.891,18.048,152.283
C04277=1097.245,256.706,423.992,177.895,18.049,152.283
C04278=1097.251,256.953,423.964,177.898,18.051,152.283
C04279=1097.256,257.202,423.937,177.901,18.052,152.282
C04280=1097.262,257.451,423.909,177.905,18.054,152.282
C04281=1097.267,257.699,423.882,177.908,18.056,152.282
C04282=1097.273,257.947,423.854,177.911,18.056,152.281
C04283=1097.279,258.196,423.827,177.915,18.058,152.281
C04284=1097.284,258.444,423.799,177.918,18.060,152.281
C04285=1097.290,258.692,423.771,177.921,18.061,152.281
C04286=1097.296,258.941,423.745,177.925,18.063,152.280
C04287=1097.302,259.189,423.716,177.928,18.065,152.280
C04288=1097.307,259.438,423.690,177.931,18.066,152.280
C04289=1097.313,259.686,423.662,177.935,18.067,152.280
C04290=1097.319,259.935,423.633,177.938,18.069,152.279
C04291=1097.324,260.183,423.607,177.941,18.070,152.279
C04292=1097.330,260.432,423.578,177.945,18.072,152.279
C04293=1097.336,260.680,423.550,177.948,18.073,152.278
C04294=1097.341,260.928,423.524,177.951,18.075,152.278
C04295=1097.347,261.177,423.495,177.955,18.076,152.278
C04296=1097.353,261.425,423.467,177.958,18.078,152.277
C04297=1097.358,261.673,423.441,177.961,18.079,152.277
C04298=1097.364,261.922,423.412,177.965,18.081,152.277
C04299=1097.370,262.170,423.384,177.968,18.083,152.277
C04300=1097.378,262.529,423.344,177.973,18.085,152.276
C04301=1097.387,262.887,423.304,177.977,18.087,152.276
C04302=1097.395,263.245,423.265,177.982,18.089,152.275
C04303=1097.404,263.603,423.224,177.987,18.091,152.275
C04304=1097.409,263.852,423.196,177.990,18.092,152.275
C04305=1097.414,264.100,423.168,177.994,18.094,152.274
C04306=1097.421,264.349,423.141,177.997,18.096,152.274
C04307=1097.427,264.597,423.113,178.001,18.098,152.274
C04308=1097.432,264.845,423.085,178.003,18.099,152.274
C04309=1097.438,265.094,423.056,178.007,18.100,152.273
C04310=1097.443,265.342,423.029,178.011,18.102,152.273
C04311=1097.449,265.591,423.000,178.013,18.104,152.273
C04312=1097.454,265.839,422.972,178.017,18.105,152.273
C04313=1097.460,266.087,422.944,178.020,18.107,152.272
C04314=1097.466,266.335,422.916,178.023,18.108,152.272
C04315=1097.471,266.583,422.888,178.027,18.110,152.272
C04316=1097.477,266.832,422.860,178.030,18.112,152.271
C04317=1097.482,267.080,422.832,178.034,18.114,152.271
C04318=1097.488,267.329,422.803,178.037,18.115,152.271
C04319=1097.494,267.577,422.775,178.040,18.116,152.271
C04320=1097.500,267.826,422.747,178.044,18.118,152.270
C04321=1097.505,268.074,422.719,178.047,18.120,152.270
C04322=1097.511,268.323,422.691,178.050,18.121,152.270
C04323=1097.516,268.571,422.663,178.054,18.123,152.270
C04324=1097.522,268.819,422.635,178.057,18.125,152.269
C04325=1097.527,269.067,422.607,178.060,18.126,152.269
C04326=1097.533,269.316,422.578,178.064,18.128,152.269
C04327=1097.539,269.564,422.550,178.067,18.130,152.269
C04328=1097.545,269.812,422.521,178.070,18.131,152.268
C04329=1097.550,270.060,422.493,178.073,18.133,152.268
C04330=1097.556,270.309,422.465,178.077,18.134,152.268
C04331=1097.562,270.557,422.437,178.080,18.136,152.268
C04332=1097.568,270.806,422.409,178.083,18.138,152.267
C04333=1097.572,271.054,422.379,178.087,18.139,152.267
C04334=1097.578,271.303,422.351,178.090,18.141,152.267
C04335=1097.584,271.551,422.323,178.094,18.143,152.267
C04336=1097.590,271.799,422.295,178.096,18.144,152.266
C04337=1097.595,272.047,422.266,178.100,18.146,152.266
C04338=1097.601,272.295,422.238,178.103,18.148,152.266
C04339=1097.607,272.544,422.209,178.107,18.150,152.266
C04340=1097.612,272.792,422.180,178.110,18.151,152.265
C04341=1097.618,273.041,422.152,178.113,18.153,152.265
C04342=1097.623,273.289,422.124,178.117,18.155,152.265
C04343=1097.630,273.537,422.095,178.120,18.157,152.265
C04344=1097.636,273.786,422.067,178.123,18.158,152.265
C04345=1097.641,274.033,422.037,178.126,18.160,152.264
C04346=1097.646,274.282,422.009,178.130,18.162,152.264
C04347=1097.652,274.530,421.981,178.133,18.163,152.264
C04348=1097.658,274.778,421.952,178.136,18.165,152.264
C04349=1097.663,275.027,421.923,178.140,18.167,152.263
C04350=1097.669,275.275,421.894,178.143,18.168,152.263
C04351=1097.675,275.524,421.866,178.147,18.170,152.263
C04352=1097.683,275.884,421.824,178.151,18.172,152.263
C04353=1097.691,276.245,421.782,178.156,18.175,152.262
C04354=1097.699,276.606,421.740,178.161,18.177,152.262
C04355=1097.707,276.968,421.698,178.166,18.180,152.262
C04356=1097.713,277.216,421.670,178.169,18.182,152.261
C04357=1097.719,277.464,421.641,178.172,18.184,152.261
C04358=1097.724,277.712,421.611,178.176,18.186,152.261
C04359=1097.730,277.960,421.583,178.179,18.187,152.261
C04360=1097.736,278.209,421.554,178.183,18.189,152.260
C04361=1097.741,278.458,421.525,178.185,18.191,152.260
C04362=1097.747,278.705,421.497,178.189,18.192,152.260
C04363=1097.752,278.954,421.467,178.192,18.194,152.260
C04364=1097.758,279.202,421.439,178.196,18.196,152.260
C04365=1097.763,279.450,421.410,178.199,18.198,152.259
C04366=1097.769,279.698,421.380,178.202,18.199,152.259
C04367=1097.776,279.946,421.351,178.205,18.202,152.259
C04368=1097.781,280.195,421.323,178.209,18.204,152.259
C04369=1097.787,280.443,421.294,178.212,18.205,152.259
C04370=1097.792,280.691,421.264,178.216,18.207,152.258
C04371=1097.798,280.939,421.235,178.219,18.209,152.258
C04372=1097.803,281.188,421.207,178.222,18.210,152.258
C04373=1097.809,281.436,421.178,178.226,18.212,152.258
C04374=1097.815,281.684,421.148,178.229,18.214,152.257
C04375=1097.821,281.932,421.119,178.233,18.216,152.257
C04376=1097.826,282.180,421.090,178.235,18.218,152.257
C04377=1097.831,282.429,421.060,178.238,18.220,152.257
C04378=1097.837,282.677,421.032,178.242,18.222,152.257
C04379=1097.843,282.926,421.002,178.245,18.223,152.256
C04380=1097.848,283.173,420.973,178.249,18.225,152.256
C04381=1097.854,283.422,420.944,178.252,18.227,152.256
C04382=1097.860,283.670,420.914,178.255,18.229,152.256
C04383=1097.866,283.918,420.885,178.258,18.231,152.256
C04384=1097.871,284.166,420.856,178.262,18.233,152.256
C04385=1097.876,284.414,420.826,178.265,18.235,152.255
C04386=1097.882,284.663,420.797,178.269,18.236,152.255
C04387=1097.888,284.911,420.767,178.272,18.239,152.255
C04388=1097.893,285.159,420.738,178.275,18.240,152.255
C04389=1097.899,285.407,420.709,178.278,18.242,152.255
C04390=1097.905,285.655,420.680,178.282,18.244,152.254
C04391=1097.910,285.904,420.650,178.285,18.246,152.254
C04392=1097.916,286.152,420.621,178.289,18.248,152.254
C04393=1097.922,286.400,420.591,178.292,18.250,152.254
C04394=1097.927,286.648,420.562,178.296,18.252,152.254
C04395=1097.933,286.896,420.532,178.298,18.254,152.254
C04396=1097.939,287.144,420.503,178.301,18.255,152.253
C04397=1097.944,287.392,420.473,178.305,18.257,152.253
C04398=1097.950,287.641,420.443,178.308,18.259,152.253
C04399=1097.956,287.889,420.414,178.312,18.261,152.253
C04400=1097.962,288.138,420.385,178.315,18.263,152.253
C04401=1097.967,288.385,420.355,178.319,18.265,152.252
C04402=1097.972,288.633,420.325,178.321,18.267,152.252
C04403=1097.979,288.881,420.296,178.325,18.269,152.252
C04404=1097.987,289.252,420.252,178.330,18.272,152.252
C04405=1097.996,289.622,420.207,178.335,18.275,152.251
C04406=1098.004,289.992,420.163,178.340,18.278,152.251
C04407=1098.012,290.364,420.119,178.345,18.280,152.251
C04408=1098.018,290.611,420.089,178.348,18.282,152.251
C04409=1098.024,290.859,420.059,178.351,18.284,152.251
C04410=1098.030,291.107,420.029,178.354,18.287,152.251
C04411=1098.035,291.356,419.999,178.358,18.288,152.250
C04412=1098.041,291.604,419.970,178.361,18.290,152.250
C04413=1098.047,291.852,419.939,178.365,18.293,152.250
C04414=1098.052,292.100,419.910,178.368,18.295,152.250
C04415=1098.058,292.348,419.879,178.371,18.296,152.250
C04416=1098.063,292.597,419.850,178.374,18.298,152.250
C04417=1098.068,292.844,419.820,178.378,18.300,152.249
C04418=1098.074,293.092,419.790,178.381,18.302,152.249
C04419=1098.080,293.341,419.760,178.384,18.304,152.249
C04420=1098.085,293.589,419.730,178.388,18.307,152.249
C04421=1098.091,293.837,419.700,178.391,18.308,152.249
C04422=1098.097,294.085,419.670,178.394,18.311,152.249
C04423=1098.102,294.333,419.640,178.398,18.313,152.248
C04424=1098.108,294.581,419.610,178.401,18.315,152.248
C04425=1098.114,294.829,419.580,178.405,18.317,152.248
C04426=1098.119,295.077,419.550,178.407,18.318,152.248
C04427=1098.125,295.325,419.520,178.410,18.321,152.248
C04428=1098.131,295.574,419.490,178.414,18.322,152.248
C04429=1098.137,295.821,419.460,178.417,18.325,152.248
C04430=1098.142,296.069,419.429,178.421,18.327,152.247
C04431=1098.148,296.318,419.400,178.424,18.329,152.247
C04432=1098.154,296.565,419.369,178.427,18.331,152.247
C04433=1098.160,296.813,419.339,178.431,18.333,152.247
C04434=1098.165,297.062,419.309,178.434,18.335,152.247
C04435=1098.171,297.310,419.279,178.437,18.337,152.247
C04436=1098.177,297.558,419.248,178.441,18.340,152.247
C04437=1098.182,297.806,419.217,178.444,18.342,152.246
C04438=1098.188,298.055,419.188,178.447,18.344,152.246
C04439=1098.194,298.302,419.157,178.451,18.346,152.246
C04440=1098.200,298.550,419.127,178.454,18.348,152.246
C04441=1098.205,298.798,419.097,178.457,18.350,152.246
C04442=1098.210,299.047,419.066,178.461,18.353,152.246
C04443=1098.216,299.295,419.036,178.463,18.354,152.246
C04444=1098.222,299.543,419.006,178.467,18.356,152.246
C04445=1098.227,299.791,418.975,178.470,18.359,152.246
C04446=1098.233,300.038,418.944,178.473,18.361,152.246
C04447=1098.238,300.286,418.914,178.476,18.363,152.245
C04448=1098.244,300.534,418.883,178.480,18.365,152.245
C04449=1098.249,300.782,418.853,178.483,18.368,152.245
C04450=1098.255,301.031,418.823,178.486,18.370,152.245
C04451=1098.260,301.279,418.792,178.489,18.372,152.245
C04452=1098.266,301.527,418.762,178.493,18.374,152.245
C04453=1098.272,301.774,418.731,178.496,18.376,152.245
C04454=1098.277,302.023,418.701,178.499,18.379,152.245
C04455=1098.282,302.270,418.670,178.503,18.381,152.245
C04456=1098.291,302.654,418.622,178.508,18.384,152.244
C04457=1098.300,303.040,418.575,178.513,18.388,152.244
C04458=1098.309,303.424,418.527,178.518,18.392,152.244
C04459=1098.317,303.808,418.480,178.523,18.395,152.244
C04460=1098.323,304.056,418.450,178.527,18.397,152.244
C04461=1098.328,304.304,418.419,178.530,18.399,152.244
C04462=1098.335,304.552,418.387,178.533,18.402,152.244
C04463=1098.340,304.800,418.356,178.536,18.404,152.244
C04464=1098.346,305.048,418.326,178.540,18.406,152.244
C04465=1098.351,305.296,418.295,178.543,18.409,152.244
C04466=1098.357,305.544,418.265,178.546,18.411,152.244
C04467=1098.362,305.792,418.234,178.550,18.413,152.243
C04468=1098.368,306.040,418.202,178.553,18.415,152.243
C04469=1098.374,306.288,418.171,178.556,18.417,152.243
C04470=1098.379,306.536,418.141,178.559,18.420,152.243
C04471=1098.384,306.784,418.110,178.562,18.422,152.243
C04472=1098.391,307.032,418.079,178.566,18.424,152.243
C04473=1098.396,307.280,418.048,178.569,18.427,152.243
C04474=1098.402,307.528,418.017,178.572,18.429,152.243
C04475=1098.407,307.775,417.986,178.575,18.431,152.243
C04476=1098.414,308.024,417.955,178.579,18.434,152.243
C04477=1098.419,308.272,417.924,178.582,18.436,152.243
C04478=1098.425,308.519,417.893,178.586,18.439,152.243
C04479=1098.430,308.767,417.862,178.589,18.441,152.242
C04480=1098.437,309.016,417.831,178.593,18.443,152.242
C04481=1098.442,309.263,417.800,178.596,18.446,152.242
C04482=1098.448,309.511,417.769,178.599,18.448,152.242
C04483=1098.454,309.759,417.737,178.602,18.450,152.242
C04484=1098.459,310.007,417.706,178.606,18.452,152.242
C04485=1098.465,310.255,417.675,178.609,18.455,152.242
C04486=1098.471,310.504,417.644,178.612,18.457,152.242
C04487=1098.477,310.751,417.613,178.615,18.459,152.242
C04488=1098.482,310.999,417.582,178.619,18.462,152.242
C04489=1098.488,311.247,417.550,178.622,18.464,152.242
C04490=1098.494,311.495,417.519,178.625,18.466,152.242
C04491=1098.500,311.743,417.487,178.628,18.469,152.242
C04492=1098.505,311.991,417.457,178.631,18.471,152.242
C04493=1098.511,312.238,417.425,178.635,18.473,152.242
C04494=1098.517,312.487,417.394,178.638,18.476,152.242
C04495=1098.523,312.734,417.363,178.641,18.478,152.242
C04496=1098.529,312.983,417.331,178.644,18.480,152.241
C04497=1098.534,313.231,417.300,178.648,18.483,152.241
C04498=1098.540,313.478,417.269,178.651,18.486,152.241
C04499=1098.546,313.727,417.238,178.655,18.488,152.241
C04500=1098.551,313.974,417.206,178.658,18.491,152.241
C04501=1098.558,314.222,417.175,178.661,18.493,152.241
C04502=1098.563,314.470,417.143,178.664,18.495,152.241
C04503=1098.569,314.719,417.112,178.668,18.498,152.241
C04504=1098.574,314.966,417.080,178.671,18.500,152.241
C04505=1098.581,315.214,417.048,178.674,18.502,152.241
C04506=1098.586,315.462,417.018,178.677,18.505,152.241
C04507=1098.592,315.710,416.986,178.680,18.507,152.241
C04508=1098.600,316.097,416.937,178.686,18.512,152.241
C04509=1098.609,316.483,416.887,178.691,18.515,152.241
C04510=1098.617,316.871,416.837,178.695,18.519,152.241
C04511=1098.626,317.258,416.788,178.701,18.524,152.241
C04512=1098.632,317.506,416.756,178.704,18.526,152.241
C04513=1098.637,317.753,416.724,178.707,18.529,152.241
C04514=1098.643,318.001,416.692,178.710,18.531,152.241
C04515=1098.649,318.249,416.660,178.713,18.534,152.241
C04516=1098.655,318.497,416.628,178.716,18.536,152.241
C04517=1098.660,318.745,416.598,178.720,18.539,152.241
C04518=1098.666,318.994,416.565,178.723,18.542,152.241
C04519=1098.671,319.241,416.534,178.727,18.544,152.241
C04520=1098.677,319.489,416.502,178.729,18.547,152.241
C04521=1098.682,319.737,416.470,178.732,18.550,152.241
C04522=1098.688,319.985,416.438,178.736,18.552,152.241
C04523=1098.693,320.233,416.406,178.739,18.555,152.241
C04524=1098.699,320.481,416.374,178.743,18.558,152.241
C04525=1098.704,320.729,416.342,178.746,18.561,152.241
C04526=1098.710,320.977,416.310,178.749,18.563,152.241
C04527=1098.716,321.224,416.278,178.752,18.566,152.242
C04528=1098.722,321.472,416.246,178.755,18.568,152.241
C04529=1098.727,321.719,416.214,178.758,18.571,152.242
C04530=1098.733,321.968,416.181,178.761,18.573,152.242
C04531=1098.738,322.215,416.150,178.765,18.576,152.242
C04532=1098.744,322.464,416.118,178.768,18.579,152.242
C04533=1098.750,322.712,416.086,178.771,18.581,152.242
C04534=1098.755,322.959,416.054,178.774,18.584,152.242
C04535=1098.762,323.207,416.021,178.777,18.587,152.242
C04536=1098.766,323.455,415.989,178.781,18.589,152.242
C04537=1098.772,323.703,415.957,178.784,18.593,152.242
C04538=1098.778,323.951,415.925,178.787,18.595,152.242
C04539=1098.784,324.198,415.893,178.791,18.598,152.242
C04540=1098.790,324.446,415.861,178.794,18.600,152.242
C04541=1098.795,324.695,415.828,178.797,18.603,152.242
C04542=1098.801,324.942,415.796,178.800,18.606,152.242
C04543=1098.807,325.190,415.764,178.804,18.609,152.242
C04544=1098.813,325.438,415.732,178.807,18.612,152.242
C04545=1098.818,325.686,415.699,178.810,18.614,152.242
C04546=1098.824,325.934,415.667,178.813,18.617,152.242
C04547=1098.830,326.182,415.635,178.816,18.619,152.242
C04548=1098.836,326.429,415.602,178.820,18.623,152.242
C04549=1098.841,326.677,415.570,178.823,18.626,152.243
C04550=1098.847,326.925,415.538,178.826,18.628,152.243
C04551=1098.853,327.173,415.505,178.829,18.631,152.243
C04552=1098.858,327.421,415.473,178.832,18.633,152.243
C04553=1098.864,327.668,415.440,178.836,18.637,152.243
C04554=1098.870,327.917,415.408,178.839,18.639,152.243
C04555=1098.876,328.164,415.375,178.842,18.642,152.243
C04556=1098.881,328.412,415.343,178.845,18.645,152.243
C04557=1098.887,328.660,415.310,178.849,18.648,152.243
C04558=1098.893,328.908,415.278,178.852,18.651,152.243
C04559=1098.899,329.156,415.245,178.854,18.653,152.243
C04560=1098.908,329.536,415.195,178.859,18.657,152.243
C04561=1098.917,329.916,415.145,178.865,18.662,152.243
C04562=1098.925,330.295,415.095,178.869,18.666,152.244
C04563=1098.934,330.675,415.045,178.874,18.671,152.244
C04564=1098.940,330.923,415.012,178.877,18.673,152.244
C04565=1098.946,331.170,414.980,178.880,18.676,152.244
C04566=1098.952,331.418,414.948,178.884,18.679,152.244
C04567=1098.957,331.666,414.914,178.887,18.682,152.244
C04568=1098.963,331.914,414.882,178.890,18.685,152.244
C04569=1098.969,332.162,414.849,178.893,18.688,152.244
C04570=1098.975,332.410,414.816,178.897,18.691,152.244
C04571=1098.981,332.658,414.783,178.900,18.694,152.244
C04572=1098.986,332.905,414.750,178.903,18.697,152.245
C04573=1098.991,333.153,414.718,178.907,18.700,152.245
C04574=1098.997,333.401,414.685,178.909,18.703,152.245
C04575=1099.003,333.649,414.652,178.912,18.706,152.245
C04576=1099.009,333.897,414.618,178.916,18.709,152.245
C04577=1099.015,334.144,414.586,178.919,18.712,152.245
C04578=1099.020,334.392,414.553,178.922,18.715,152.245
C04579=1099.025,334.640,414.520,178.925,18.718,152.246
C04580=1099.032,334.888,414.487,178.929,18.721,152.246
C04581=1099.037,335.136,414.454,178.932,18.724,152.246
C04582=1099.043,335.383,414.421,178.934,18.727,152.246
C04583=1099.049,335.631,414.388,178.938,18.730,152.246
C04584=1099.055,335.879,414.355,178.941,18.733,152.246
C04585=1099.060,336.126,414.322,178.944,18.736,152.246
C04586=1099.065,336.374,414.288,178.948,18.740,152.247
C04587=1099.071,336.622,414.256,178.951,18.742,152.247
C04588=1099.077,336.870,414.222,178.953,18.746,152.247
C04589=1099.083,337.117,414.189,178.957,18.749,152.247
C04590=1099.089,337.365,414.156,178.960,18.752,152.247
C04591=1099.094,337.613,414.123,178.963,18.755,152.247
C04592=1099.100,337.861,414.089,178.967,18.758,152.247
C04593=1099.105,338.109,414.056,178.969,18.761,152.248
C04594=1099.112,338.356,414.023,178.972,18.764,152.248
C04595=1099.117,338.604,413.990,178.976,18.768,152.248
C04596=1099.123,338.852,413.956,178.979,18.771,152.248
C04597=1099.129,339.099,413.923,178.982,18.774,152.248
C04598=1099.134,339.347,413.889,178.985,18.777,152.249
C04599=1099.140,339.595,413.856,178.988,18.780,152.249
C04600=1099.146,339.842,413.824,178.991,18.784,152.249
C04601=1099.151,340.090,413.790,178.995,18.787,152.249
C04602=1099.157,340.337,413.756,178.997,18.790,152.249
C04603=1099.163,340.585,413.723,179.001,18.794,152.250
C04604=1099.168,340.833,413.690,179.004,18.797,152.250
C04605=1099.174,341.081,413.656,179.007,18.800,152.250
C04606=1099.180,341.328,413.622,179.010,18.804,152.250
C04607=1099.185,341.576,413.589,179.013,18.806,152.250
C04608=1099.191,341.824,413.555,179.017,18.810,152.251
C04609=1099.196,342.071,413.521,179.019,18.813,152.251
C04610=1099.202,342.319,413.488,179.022,18.816,152.251
C04611=1099.208,342.567,413.455,179.026,18.820,152.251
C04612=1099.217,342.941,413.404,179.030,18.824,152.252
C04613=1099.226,343.315,413.353,179.035,18.830,152.252
C04614=1099.234,343.688,413.302,179.040,18.835,152.252
C04615=1099.243,344.063,413.251,179.044,18.839,152.253
C04616=1099.249,344.310,413.217,179.048,18.843,152.253
C04617=1099.254,344.558,413.184,179.051,18.846,152.253
C04618=1099.260,344.805,413.150,179.054,18.850,152.253
C04619=1099.266,345.053,413.117,179.057,18.853,152.253
C04620=1099.272,345.300,413.083,179.061,18.857,152.254
C04621=1099.277,345.548,413.049,179.063,18.860,152.254
C04622=1099.283,345.795,413.015,179.066,18.863,152.254
C04623=1099.289,346.044,412.981,179.070,18.867,152.254
C04624=1099.294,346.292,412.947,179.072,18.870,152.255
C04625=1099.300,346.540,412.914,179.076,18.874,152.255
C04626=1099.306,346.787,412.879,179.078,18.877,152.255
C04627=1099.312,347.034,412.845,179.082,18.881,152.256
C04628=1099.317,347.282,412.812,179.085,18.884,152.256
C04629=1099.323,347.529,412.778,179.088,18.888,152.256
C04630=1099.328,347.777,412.743,179.091,18.891,152.256
C04631=1099.334,348.025,412.710,179.095,18.895,152.257
C04632=1099.340,348.273,412.676,179.097,18.898,152.257
C04633=1099.346,348.520,412.642,179.101,18.902,152.257
C04634=1099.351,348.768,412.607,179.103,18.905,152.257
C04635=1099.357,349.016,412.574,179.107,18.909,152.258
C04636=1099.362,349.263,412.540,179.110,18.912,152.258
C04637=1099.368,349.510,412.505,179.113,18.917,152.258
C04638=1099.374,349.758,412.470,179.116,18.920,152.259
C04639=1099.380,350.006,412.436,179.119,18.923,152.259
C04640=1099.386,350.253,412.402,179.122,18.927,152.259
C04641=1099.391,350.501,412.369,179.125,18.931,152.260
C04642=1099.396,350.748,412.334,179.128,18.934,152.260
C04643=1099.402,350.996,412.300,179.131,18.938,152.260
C04644=1099.409,351.244,412.266,179.134,18.941,152.260
C04645=1099.414,351.491,412.231,179.138,18.945,152.261
C04646=1099.420,351.739,412.197,179.140,18.949,152.261
C04647=1099.426,351.986,412.163,179.144,18.952,152.261
C04648=1099.431,352.234,412.128,179.146,18.956,152.262
C04649=1099.437,352.481,412.094,179.150,18.960,152.262
C04650=1099.443,352.729,412.060,179.152,18.963,152.262
C04651=1099.448,352.976,412.025,179.156,18.967,152.263
C04652=1099.455,353.224,411.991,179.158,18.971,152.263
C04653=1099.460,353.472,411.956,179.162,18.974,152.263
C04654=1099.466,353.719,411.922,179.164,18.978,152.264
C04655=1099.472,353.967,411.888,179.168,18.982,152.264
C04656=1099.477,354.215,411.853,179.171,18.986,152.264
C04657=1099.483,354.462,411.819,179.174,18.990,152.265
C04658=1099.489,354.709,411.784,179.177,18.993,152.265
C04659=1099.494,354.956,411.750,179.180,18.997,152.265
C04660=1099.500,355.205,411.715,179.183,19.001,152.266
C04661=1099.506,355.452,411.681,179.186,19.005,152.266
C04662=1099.511,355.700,411.646,179.189,19.008,152.267
C04663=1099.516,355.947,411.611,179.192,19.013,152.267
C04664=1099.526,356.323,411.558,179.197,19.019,152.268
C04665=1099.534,356.699,411.506,179.202,19.024,152.268
C04666=1099.543,357.075,411.453,179.206,19.030,152.269
C04667=1099.552,357.451,411.401,179.211,19.036,152.269
C04668=1099.557,357.699,411.366,179.213,19.040,152.270
C04669=1099.564,357.946,411.331,179.217,19.044,152.270
C04670=1099.569,358.194,411.296,179.219,19.047,152.270
C04671=1099.574,358.442,411.261,179.223,19.051,152.271
C04672=1099.581,358.689,411.226,179.226,19.056,152.271
C04673=1099.586,358.937,411.191,179.228,19.059,152.272
C04674=1099.592,359.184,411.156,179.232,19.063,152.272
C04675=1099.598,359.431,411.122,179.234,19.067,152.272
C04676=1099.604,359.679,411.086,179.237,19.071,152.273
C04677=1099.610,359.926,411.052,179.241,19.076,152.273
C04678=1099.616,360.174,411.016,179.243,19.079,152.274
C04679=1099.621,360.421,410.982,179.246,19.083,152.274
C04680=1099.626,360.668,410.946,179.250,19.088,152.275
C04681=1099.633,360.916,410.912,179.252,19.091,152.275
C04682=1099.638,361.163,410.877,179.255,19.096,152.276
C04683=1099.643,361.411,410.842,179.259,19.100,152.276
C04684=1099.649,361.659,410.806,179.261,19.104,152.276
C04685=1099.655,361.906,410.772,179.264,19.108,152.277
C04686=1099.661,362.154,410.736,179.267,19.112,152.277
C04687=1099.666,362.400,410.701,179.270,19.116,152.278
C04688=1099.672,362.649,410.666,179.273,19.120,152.278
C04689=1099.678,362.895,410.631,179.276,19.125,152.279
C04690=1099.684,363.142,410.596,179.279,19.128,152.279
C04691=1099.690,363.391,410.561,179.282,19.133,152.280
C04692=1099.695,363.638,410.526,179.285,19.137,152.280
C04693=1099.701,363.885,410.490,179.288,19.141,152.281
C04694=1099.706,364.132,410.454,179.291,19.145,152.281
C04695=1099.713,364.380,410.420,179.294,19.150,152.282
C04696=1099.718,364.627,410.385,179.296,19.153,152.282
C04697=1099.724,364.875,410.349,179.300,19.158,152.283
C04698=1099.730,365.122,410.314,179.303,19.162,152.283
C04699=1099.736,365.370,410.278,179.306,19.167,152.284
C04700=1099.741,365.617,410.243,179.308,19.171,152.284
C04701=1099.747,365.865,410.207,179.311,19.175,152.284
C04702=1099.752,366.112,410.172,179.315,19.179,152.285
C04703=1099.758,366.360,410.136,179.318,19.184,152.286
C04704=1099.764,366.607,410.101,179.320,19.188,152.286
C04705=1099.770,366.854,410.065,179.323,19.192,152.287
C04706=1099.775,367.101,410.030,179.326,19.197,152.287
C04707=1099.781,367.349,409.994,179.329,19.201,152.288
C04708=1099.787,367.596,409.959,179.332,19.205,152.288
C04709=1099.793,367.843,409.923,179.335,19.210,152.289
C04710=1099.798,368.090,409.888,179.338,19.214,152.289
C04711=1099.804,368.338,409.852,179.341,19.219,152.290
C04712=1099.810,368.585,409.817,179.343,19.223,152.290
C04713=1099.816,368.833,409.781,179.346,19.227,152.291
C04714=1099.821,369.080,409.746,179.349,19.232,152.292
C04715=1099.827,369.327,409.710,179.352,19.237,152.292
C04716=1099.833,369.605,409.669,179.355,19.242,152.293
C04717=1099.840,369.881,409.630,179.358,19.246,152.293
C04718=1099.846,370.158,409.589,179.362,19.252,152.294
C04719=1099.853,370.435,409.549,179.365,19.256,152.295
C04720=1099.858,370.682,409.513,179.368,19.261,152.295
C04721=1099.864,370.930,409.477,179.371,19.266,152.296
C04722=1099.869,371.177,409.442,179.373,19.270,152.296
C04723=1099.875,371.425,409.406,179.376,19.274,152.297
C04724=1099.882,371.672,409.370,179.379,19.279,152.298
C04725=1099.887,371.919,409.335,179.382,19.284,152.298
C04726=1099.893,372.167,409.298,179.385,19.289,152.299
C04727=1099.899,372.414,409.262,179.388,19.293,152.299
C04728=1099.904,372.661,409.226,179.391,19.298,152.300
C04729=1099.910,372.908,409.191,179.394,19.302,152.301
C04730=1099.916,373.155,409.155,179.396,19.307,152.301
C04731=1099.922,373.402,409.119,179.400,19.312,152.302
C04732=1099.927,373.650,409.083,179.403,19.316,152.302
C04733=1099.934,373.897,409.046,179.405,19.321,152.303
C04734=1099.939,374.144,409.011,179.408,19.325,152.304
C04735=1099.946,374.391,408.974,179.411,19.330,152.304
C04736=1099.951,374.639,408.938,179.413,19.335,152.305
C04737=1099.957,374.886,408.902,179.417,19.340,152.306
C04738=1099.963,375.134,408.866,179.419,19.345,152.306
C04739=1099.968,375.381,408.829,179.422,19.350,152.307
C04740=1099.974,375.628,408.794,179.425,19.355,152.308
C04741=1099.979,375.875,408.757,179.427,19.359,152.308
C04742=1099.985,376.123,408.721,179.430,19.364,152.309
C04743=1099.990,376.370,408.684,179.433,19.369,152.310
C04744=1099.996,376.617,408.649,179.436,19.374,152.310
C04745=1100.003,376.864,408.612,179.439,19.379,152.311
C04746=1100.008,377.111,408.575,179.442,19.384,152.312
C04747=1100.014,377.359,408.540,179.445,19.389,152.313
C04748=1100.019,377.606,408.503,179.447,19.393,152.313
C04749=1100.025,377.852,408.467,179.450,19.398,152.314
C04750=1100.030,378.100,408.430,179.453,19.403,152.315
C04751=1100.037,378.347,408.394,179.456,19.408,152.315
C04752=1100.042,378.595,408.357,179.459,19.413,152.316
C04753=1100.048,378.841,408.321,179.461,19.418,152.317
C04754=1100.053,379.089,408.284,179.464,19.423,152.317
C04755=1100.060,379.336,408.248,179.466,19.428,152.318
C04756=1100.065,379.583,408.211,179.469,19.433,152.319
C04757=1100.071,379.831,408.174,179.472,19.438,152.320
C04758=1100.076,380.077,408.138,179.475,19.443,152.320
C04759=1100.083,380.325,408.102,179.478,19.448,152.321
C04760=1100.091,380.686,408.048,179.482,19.455,152.322
C04761=1100.100,381.047,407.995,179.486,19.463,152.323
C04762=1100.108,381.409,407.941,179.490,19.471,152.324
C04763=1100.117,381.770,407.887,179.494,19.478,152.326
C04764=1100.123,382.017,407.851,179.497,19.483,152.326
C04765=1100.128,382.264,407.814,179.499,19.489,152.327
C04766=1100.134,382.511,407.778,179.502,19.493,152.328
C04767=1100.140,382.759,407.741,179.505,19.499,152.329
C04768=1100.150,383.176,407.678,179.510,19.508,152.330
C04769=1100.160,383.595,407.615,179.514,19.517,152.331
C04770=1100.169,384.013,407.553,179.519,19.526,152.333
C04771=1100.178,384.431,407.491,179.523,19.535,152.334
C04772=1100.184,384.678,407.454,179.526,19.540,152.335
C04773=1100.190,384.925,407.416,179.528,19.545,152.336
C04774=1100.195,385.172,407.379,179.531,19.551,152.337
C04775=1100.202,385.420,407.343,179.534,19.556,152.338
C04776=1100.207,385.667,407.306,179.537,19.562,152.338
C04777=1100.213,385.914,407.269,179.540,19.568,152.339
C04778=1100.218,386.160,407.231,179.542,19.573,152.340
C04779=1100.224,386.408,407.194,179.545,19.578,152.341
C04780=1100.230,386.655,407.157,179.547,19.584,152.342
C04781=1100.236,386.901,407.120,179.550,19.589,152.343
C04782=1100.242,387.149,407.083,179.553,19.595,152.344
C04783=1100.247,387.396,407.046,179.555,19.600,152.345
C04784=1100.253,387.643,407.008,179.558,19.606,152.345
C04785=1100.259,387.890,406.971,179.560,19.611,152.346
C04786=1100.264,388.138,406.934,179.564,19.617,152.347
C04787=1100.270,388.384,406.896,179.566,19.623,152.348
C04788=1100.277,388.631,406.860,179.569,19.629,152.349
C04789=1100.283,388.878,406.822,179.572,19.634,152.350
C04790=1100.288,389.126,406.785,179.574,19.640,152.351
C04791=1100.294,389.372,406.747,179.577,19.645,152.352
C04792=1100.300,389.620,406.710,179.579,19.651,152.353
C04793=1100.306,389.866,406.673,179.582,19.657,152.354
C04794=1100.311,390.114,406.636,179.585,19.663,152.355
C04795=1100.317,390.361,406.598,179.588,19.668,152.355
C04796=1100.323,390.608,406.561,179.590,19.674,152.356
C04797=1100.329,390.855,406.523,179.592,19.680,152.357
C04798=1100.335,391.101,406.485,179.595,19.685,152.358
C04799=1100.340,391.349,406.448,179.597,19.691,152.359
C04800=1100.346,391.595,406.411,179.601,19.697,152.360
C04801=1100.352,391.843,406.374,179.603,19.703,152.361
C04802=1100.358,392.090,406.335,179.606,19.709,152.362
C04803=1100.364,392.337,406.298,179.608,19.714,152.363
C04804=1100.370,392.584,406.261,179.610,19.720,152.364
C04805=1100.376,392.831,406.223,179.614,19.726,152.365
C04806=1100.381,393.078,406.185,179.616,19.732,152.366
C04807=1100.387,393.325,406.147,179.619,19.738,152.367
C04808=1100.393,393.572,406.110,179.621,19.744,152.368
C04809=1100.398,393.819,406.072,179.623,19.750,152.369
C04810=1100.404,394.066,406.034,179.626,19.756,152.370
C04811=1100.411,394.313,405.996,179.629,19.762,152.371
C04812=1100.416,394.560,405.958,179.631,19.768,152.372
C04813=1100.422,394.807,405.921,179.633,19.774,152.373
C04814=1100.427,395.054,405.883,179.637,19.780,152.374
C04815=1100.433,395.301,405.845,179.639,19.786,152.375
C04816=1100.439,395.548,405.807,179.641,19.792,152.377
C04817=1100.446,395.795,405.769,179.644,19.798,152.378
C04818=1100.451,396.042,405.731,179.647,19.805,152.379
C04819=1100.457,396.289,405.693,179.649,19.811,152.380
C04820=1100.461,396.504,405.660,179.652,19.816,152.381
C04821=1100.467,396.720,405.627,179.653,19.822,152.382
C04822=1100.471,396.935,405.594,179.656,19.827,152.383
C04823=1100.477,397.151,405.561,179.657,19.833,152.384
C04824=1100.481,397.366,405.528,179.660,19.838,152.385
C04825=1100.486,397.581,405.494,179.663,19.844,152.386
C04826=1100.492,397.796,405.461,179.664,19.849,152.387
C04827=1100.496,398.012,405.428,179.667,19.855,152.388
C04828=1100.503,398.259,405.390,179.669,19.861,152.389
C04829=1100.508,398.506,405.352,179.671,19.867,152.390
C04830=1100.514,398.753,405.314,179.674,19.874,152.391
C04831=1100.520,399.000,405.276,179.676,19.880,152.392
C04832=1100.526,399.247,405.237,179.679,19.887,152.393
C04833=1100.532,399.493,405.199,179.682,19.893,152.394
C04834=1100.537,399.741,405.161,179.684,19.899,152.396
C04835=1100.544,399.988,405.123,179.687,19.906,152.397
C04836=1100.549,400.235,405.084,179.689,19.912,152.398
C04837=1100.555,400.481,405.046,179.691,19.919,152.399
C04838=1100.560,400.728,405.007,179.694,19.926,152.400
C04839=1100.567,400.976,404.969,179.696,19.932,152.401
C04840=1100.572,401.223,404.931,179.699,19.939,152.403
C04841=1100.578,401.469,404.892,179.701,19.945,152.404
C04842=1100.584,401.717,404.854,179.703,19.952,152.405
C04843=1100.590,401.963,404.816,179.706,19.959,152.406
C04844=1100.595,402.210,404.777,179.708,19.965,152.408
C04845=1100.601,402.458,404.738,179.711,19.972,152.409
C04846=1100.607,402.704,404.700,179.713,19.979,152.410
C04847=1100.613,402.951,404.661,179.716,19.986,152.411
C04848=1100.619,403.198,404.623,179.718,19.992,152.413
C04849=1100.624,403.445,404.584,179.720,19.999,152.414
C04850=1100.630,403.692,404.545,179.723,20.006,152.415
C04851=1100.636,403.938,404.507,179.725,20.012,152.416
C04852=1100.642,404.186,404.468,179.728,20.020,152.418
C04853=1100.648,404.432,404.430,179.730,20.026,152.419
C04854=1100.653,404.679,404.391,179.733,20.033,152.420
C04855=1100.659,404.927,404.352,179.735,20.040,152.422
C04856=1100.665,405.174,404.314,179.738,20.047,152.423
C04857=1100.671,405.420,404.275,179.740,20.054,152.424
C04858=1100.677,405.667,404.237,179.742,20.061,152.425
C04859=1100.683,405.915,404.197,179.745,20.068,152.427
C04860=1100.688,406.161,404.158,179.747,20.075,152.428
C04861=1100.695,406.408,404.120,179.750,20.082,152.429
C04862=1100.700,406.655,404.081,179.752,20.089,152.431
C04863=1100.706,406.901,404.042,179.754,20.097,152.432
C04864=1100.711,407.149,404.003,179.756,20.104,152.434
C04865=1100.717,407.396,403.964,179.759,20.111,152.435
C04866=1100.724,407.642,403.925,179.762,20.118,152.436
C04867=1100.729,407.889,403.886,179.763,20.125,152.438
C04868=1100.735,408.137,403.847,179.766,20.132,152.439
C04869=1100.740,408.383,403.808,179.768,20.139,152.440
C04870=1100.746,408.630,403.769,179.771,20.147,152.442
C04871=1100.752,408.877,403.730,179.773,20.154,152.443
C04872=1100.758,409.124,403.690,179.775,20.161,152.445
C04873=1100.763,409.370,403.651,179.778,20.169,152.446
C04874=1100.769,409.618,403.613,179.780,20.177,152.448
C04875=1100.775,409.864,403.574,179.782,20.184,152.449
C04876=1100.780,410.079,403.540,179.784,20.190,152.450
C04877=1100.785,410.295,403.505,179.786,20.197,152.452
C04878=1100.790,410.511,403.470,179.788,20.204,152.453
C04879=1100.796,410.726,403.436,179.790,20.210,152.454
C04880=1100.801,410.941,403.402,179.792,20.217,152.455
C04881=1100.806,411.157,403.367,179.794,20.223,152.457
C04882=1100.811,411.371,403.334,179.796,20.230,152.458
C04883=1100.815,411.587,403.299,179.798,20.236,152.459
C04884=1100.822,411.834,403.260,179.801,20.244,152.461
C04885=1100.828,412.081,403.220,179.804,20.252,152.462
C04886=1100.833,412.327,403.181,179.805,20.259,152.464
C04887=1100.839,412.575,403.142,179.808,20.267,152.465
C04888=1100.845,412.821,403.103,179.810,20.275,152.467
C04889=1100.851,413.068,403.063,179.813,20.283,152.468
C04890=1100.857,413.315,403.023,179.815,20.290,152.470
C04891=1100.862,413.561,402.983,179.817,20.298,152.471
C04892=1100.868,413.809,402.944,179.819,20.306,152.473
C04893=1100.874,414.056,402.905,179.822,20.314,152.475
C04894=1100.880,414.302,402.865,179.824,20.322,152.476
C04895=1100.886,414.549,402.825,179.827,20.330,152.478
C04896=1100.892,414.796,402.786,179.828,20.337,152.479
C04897=1100.897,415.042,402.747,179.831,20.345,152.481
C04898=1100.904,415.289,402.707,179.833,20.353,152.483
C04899=1100.910,415.536,402.667,179.835,20.361,152.484
C04900=1100.915,415.783,402.627,179.838,20.369,152.486
C04901=1100.921,416.029,402.587,179.840,20.377,152.487
C04902=1100.927,416.276,402.548,179.843,20.385,152.489
C04903=1100.933,416.523,402.508,179.845,20.394,152.491
C04904=1100.939,416.769,402.469,179.846,20.401,152.492
C04905=1100.944,417.016,402.428,179.849,20.409,152.494
C04906=1100.951,417.263,402.389,179.851,20.418,152.496
C04907=1100.957,417.510,402.349,179.853,20.426,152.497
C04908=1100.962,417.756,402.309,179.855,20.434,152.499
C04909=1100.968,418.003,402.269,179.858,20.443,152.501
C04910=1100.973,418.250,402.229,179.860,20.451,152.502
C04911=1100.979,418.496,402.189,179.862,20.459,152.504
C04912=1100.986,418.743,402.149,179.864,20.468,152.506
C04913=1100.991,418.990,402.109,179.867,20.476,152.508
C04914=1100.997,419.237,402.069,179.869,20.485,152.509
C04915=1101.004,419.483,402.028,179.871,20.493,152.511
C04916=1101.008,419.730,401.989,179.873,20.502,152.513
C04917=1101.015,419.976,401.949,179.875,20.510,152.514
C04918=1101.020,420.223,401.908,179.877,20.519,152.516
C04919=1101.026,420.470,401.868,179.880,20.527,152.518
C04920=1101.032,420.717,401.828,179.882,20.536,152.520
C04921=1101.038,420.963,401.788,179.884,20.544,152.522
C04922=1101.044,421.210,401.747,179.886,20.553,152.523
C04923=1101.050,421.456,401.707,179.888,20.562,152.525
C04924=1101.056,421.703,401.667,179.891,20.571,152.527
C04925=1101.062,421.950,401.626,179.893,20.580,152.529
C04926=1101.068,422.197,401.587,179.895,20.588,152.531
C04927=1101.073,422.443,401.546,179.897,20.597,152.533
C04928=1101.079,422.690,401.506,179.899,20.606,152.534
C04929=1101.085,422.936,401.465,179.902,20.615,152.536
C04930=1101.091,423.183,401.425,179.904,20.623,152.538
C04931=1101.097,423.430,401.385,179.905,20.632,152.540
C04932=1101.103,423.652,401.347,179.908,20.641,152.542
C04933=1101.107,423.874,401.311,179.909,20.648,152.543
C04934=1101.113,424.096,401.275,179.912,20.657,152.545
C04935=1101.118,424.318,401.238,179.914,20.665,152.547
C04936=1101.123,424.540,401.202,179.915,20.673,152.549
C04937=1101.129,424.763,401.165,179.917,20.682,152.550
C04938=1101.134,424.985,401.128,179.919,20.690,152.552
C04939=1101.139,425.207,401.092,179.921,20.698,152.554
C04940=1101.145,425.453,401.051,179.923,20.707,152.556
C04941=1101.150,425.700,401.011,179.925,20.716,152.558
C04942=1101.157,425.946,400.970,179.927,20.726,152.560
C04943=1101.163,426.193,400.929,179.929,20.735,152.562
C04944=1101.168,426.440,400.888,179.931,20.744,152.564
C04945=1101.174,426.687,400.848,179.933,20.754,152.566
C04946=1101.181,426.933,400.807,179.936,20.763,152.568
C04947=1101.186,427.179,400.766,179.938,20.773,152.570
C04948=1101.192,427.426,400.725,179.940,20.782,152.572
C04949=1101.198,427.672,400.684,179.941,20.791,152.574
C04950=1101.203,427.919,400.643,179.944,20.801,152.576
C04951=1101.210,428.165,400.602,179.946,20.811,152.578
C04952=1101.216,428.412,400.561,179.947,20.820,152.580
C04953=1101.221,428.659,400.521,179.950,20.830,152.582
C04954=1101.227,428.905,400.479,179.952,20.840,152.584
C04955=1101.233,429.152,400.439,179.953,20.849,152.587
C04956=1101.240,429.398,400.398,179.956,20.859,152.589
C04957=1101.245,429.645,400.357,179.958,20.869,152.591
C04958=1101.251,429.891,400.315,179.959,20.878,152.593
C04959=1101.257,430.137,400.274,179.962,20.889,152.595
C04960=1101.263,430.384,400.233,179.963,20.898,152.597
C04961=1101.269,430.630,400.192,179.965,20.908,152.599
C04962=1101.274,430.877,400.151,179.968,20.918,152.602
C04963=1101.280,431.123,400.110,179.969,20.928,152.604
C04964=1101.286,431.369,400.068,179.972,20.938,152.606
C04965=1101.292,431.615,400.027,179.973,20.948,152.608
C04966=1101.298,431.862,399.986,179.976,20.959,152.610
C04967=1101.304,432.108,399.945,179.977,20.968,152.613
C04968=1101.310,432.355,399.903,179.979,20.978,152.615
C04969=1101.316,432.602,399.861,179.981,20.989,152.617
C04970=1101.322,432.848,399.820,179.983,20.999,152.619
C04971=1101.328,433.095,399.779,179.985,21.010,152.622
C04972=1101.334,433.341,399.738,179.986,21.020,152.624
C04973=1101.340,433.587,399.696,179.989,21.030,152.626
C04974=1101.345,433.833,399.654,179.990,21.040,152.629
C04975=1101.351,434.080,399.613,179.992,21.051,152.631
C04976=1101.357,434.326,399.571,179.994,21.061,152.633
C04977=1101.363,434.572,399.530,179.996,21.072,152.636
C04978=1101.369,434.819,399.487,179.998,21.082,152.638
C04979=1101.375,435.065,399.446,180.000,21.093,152.641
C04980=1101.381,435.312,399.404,-179.998,21.104,152.643
C04981=1101.387,435.558,399.363,-179.997,21.115,152.645
C04982=1101.393,435.804,399.321,-179.995,21.125,152.648
C04983=1101.398,436.051,399.279,-179.993,21.136,152.650
C04984=1101.404,436.297,399.238,-179.991,21.147,152.653
C04985=1101.410,436.544,399.196,-179.990,21.157,152.655
C04986=1101.415,436.790,399.154,-179.988,21.169,152.657
C04987=1101.422,437.036,399.112,-179.986,21.180,152.660
C04988=1101.430,437.406,399.049,-179.983,21.196,152.664
C04989=1101.440,437.776,398.986,-179.980,21.213,152.667
C04990=1101.449,438.147,398.923,-179.978,21.230,152.671
C04991=1101.458,438.517,398.860,-179.975,21.246,152.675
C04992=1101.463,438.763,398.818,-179.974,21.257,152.678
C04993=1101.469,439.010,398.776,-179.972,21.268,152.680
C04994=1101.476,439.256,398.734,-179.970,21.280,152.683
C04995=1101.482,439.502,398.692,-179.969,21.290,152.685
C04996=1101.487,439.748,398.650,-179.967,21.302,152.688
C04997=1101.494,439.995,398.608,-179.965,21.314,152.690
C04998=1101.500,440.240,398.566,-179.963,21.325,152.693
C04999=1101.505,440.487,398.524,-179.962,21.336,152.696
C05000=1101.512,440.733,398.481,-179.960,21.348,152.698
C05001=1101.517,440.980,398.439,-179.958,21.360,152.701
C05002=1101.523,441.225,398.397,-179.956,21.371,152.704
C05003=1101.529,441.472,398.355,-179.955,21.383,152.706
C05004=1101.535,441.718,398.312,-179.954,21.395,152.709
C05005=1101.541,441.964,398.269,-179.952,21.407,152.712
C05006=1101.546,442.210,398.227,-179.950,21.418,152.715
C05007=1101.553,442.457,398.185,-179.948,21.430,152.717
C05008=1101.559,442.703,398.142,-179.947,21.442,152.720
C05009=1101.565,442.948,398.100,-179.946,21.454,152.723
C05010=1101.571,443.195,398.057,-179.944,21.466,152.726
C05011=1101.576,443.441,398.015,-179.942,21.478,152.729
C05012=1101.582,443.687,397.973,-179.941,21.490,152.731
C05013=1101.588,443.934,397.929,-179.940,21.502,152.734
C05014=1101.594,444.179,397.887,-179.938,21.514,152.737
C05015=1101.601,444.426,397.845,-179.937,21.526,152.740
C05016=1101.606,444.672,397.802,-179.937,21.538,152.743
C05017=1101.612,444.919,397.759,-179.936,21.550,152.746
C05018=1101.618,445.164,397.717,-179.935,21.562,152.749
C05019=1101.624,445.410,397.674,-179.935,21.574,152.752
C05020=1101.630,445.657,397.631,-179.934,21.586,152.755
C05021=1101.636,445.903,397.588,-179.934,21.598,152.758
C05022=1101.642,446.149,397.546,-179.935,21.610,152.761
C05023=1101.648,446.395,397.503,-179.934,21.622,152.764
C05024=1101.654,446.642,397.460,-179.934,21.634,152.767
C05025=1101.660,446.887,397.417,-179.935,21.645,152.770
C05026=1101.666,447.134,397.374,-179.935,21.657,152.773
C05027=1101.671,447.380,397.331,-179.935,21.669,152.776
C05028=1101.677,447.627,397.288,-179.936,21.681,152.779
C05029=1101.683,447.872,397.245,-179.937,21.693,152.782
C05030=1101.690,448.119,397.203,-179.938,21.705,152.785
C05031=1101.695,448.365,397.160,-179.939,21.716,152.789
C05032=1101.702,448.611,397.116,-179.940,21.728,152.792
C05033=1101.707,448.856,397.073,-179.941,21.740,152.795
C05034=1101.713,449.103,397.030,-179.942,21.751,152.798
C05035=1101.719,449.350,396.987,-179.944,21.763,152.801
C05036=1101.725,449.596,396.944,-179.945,21.775,152.805
C05037=1101.730,449.841,396.901,-179.946,21.787,152.808
C05038=1101.737,450.087,396.857,-179.949,21.798,152.811
C05039=1101.744,450.334,396.815,-179.950,21.810,152.814
C05040=1101.344,450.326,396.674,179.981,22.033,152.882
C05041=1101.337,450.080,396.716,179.983,22.022,152.878
C05042=1101.331,449.833,396.759,179.984,22.010,152.875
C05043=1101.325,449.588,396.803,179.986,21.998,152.872
C05044=1101.319,449.341,396.846,179.988,21.987,152.869
C05045=1101.314,449.095,396.889,179.989,21.975,152.866
C05046=1101.307,448.849,396.933,179.990,21.963,152.862
C05047=1101.302,448.604,396.975,179.991,21.951,152.859
C05048=1101.296,448.357,397.018,179.992,21.939,152.856
C05049=1101.290,448.110,397.062,179.993,21.927,152.853
C05050=1101.284,447.864,397.104,179.994,21.916,152.850
C05051=1101.278,447.618,397.147,179.995,21.903,152.846
C05052=1101.271,447.373,397.190,179.995,21.891,152.843
C05053=1101.265,447.126,397.233,179.996,21.880,152.840
C05054=1101.260,446.880,397.276,179.996,21.868,152.837
C05055=1101.254,446.634,397.319,179.997,21.856,152.834
C05056=1101.248,446.388,397.362,179.997,21.844,152.831
C05057=1101.242,446.141,397.405,179.996,21.831,152.828
C05058=1101.236,445.895,397.448,179.997,21.820,152.825
C05059=1101.230,445.649,397.491,179.996,21.807,152.822
C05060=1101.224,445.403,397.533,179.996,21.796,152.819
C05061=1101.218,445.157,397.576,179.995,21.784,152.816
C05062=1101.212,444.911,397.619,179.994,21.772,152.813
C05063=1101.206,444.664,397.662,179.994,21.759,152.810
C05064=1101.200,444.419,397.705,179.993,21.748,152.807
C05065=1101.194,444.172,397.748,179.991,21.735,152.804
C05066=1101.188,443.926,397.790,179.990,21.723,152.801
C05067=1101.182,443.681,397.833,179.989,21.711,152.798
C05068=1101.176,443.434,397.876,179.988,21.699,152.796
C05069=1101.171,443.188,397.919,179.986,21.687,152.793
C05070=1101.164,442.941,397.960,179.984,21.675,152.790
C05071=1101.159,442.695,398.003,179.982,21.663,152.787
C05072=1101.152,442.450,398.045,179.981,21.650,152.784
C05073=1101.146,442.203,398.088,179.979,21.638,152.782
C05074=1101.141,441.957,398.130,179.978,21.627,152.779
C05075=1101.135,441.711,398.173,179.976,21.615,152.776
C05076=1101.129,441.464,398.216,179.974,21.603,152.773
C05077=1101.122,441.219,398.258,179.972,21.591,152.771
C05078=1101.116,440.972,398.300,179.970,21.580,152.768
C05079=1101.110,440.726,398.343,179.969,21.568,152.765
C05080=1101.105,440.479,398.385,179.967,21.556,152.763
C05081=1101.099,440.234,398.427,179.965,21.545,152.760
C05082=1101.093,439.987,398.469,179.963,21.533,152.757
C05083=1101.087,439.741,398.511,179.962,21.522,152.755
C05084=1101.080,439.496,398.554,179.960,21.510,152.752
C05085=1101.075,439.248,398.596,179.958,21.499,152.750
C05086=1101.069,439.002,398.637,179.957,21.488,152.747
C05087=1101.063,438.756,398.680,179.955,21.476,152.744
C05088=1101.057,438.509,398.722,179.953,21.465,152.742
C05089=1101.048,438.146,398.784,179.950,21.448,152.738
C05090=1101.039,437.783,398.846,179.948,21.432,152.734
C05091=1101.030,437.419,398.908,179.945,21.416,152.731
C05092=1101.021,437.057,398.970,179.942,21.400,152.727
C05093=1101.016,436.810,399.012,179.940,21.388,152.724
C05094=1101.009,436.563,399.054,179.939,21.378,152.722
C05095=1101.003,436.317,399.095,179.937,21.367,152.720
C05096=1100.998,436.071,399.137,179.935,21.356,152.717
C05097=1100.992,435.825,399.180,179.933,21.345,152.715
C05098=1100.986,435.579,399.221,179.931,21.334,152.712
C05099=1100.980,435.333,399.263,179.930,21.323,152.710
C05100=1100.974,435.086,399.304,179.927,21.312,152.707
C05101=1100.968,434.839,399.346,179.926,21.302,152.705
C05102=1100.962,434.593,399.388,179.924,21.291,152.703
C05103=1100.956,434.347,399.429,179.922,21.281,152.700
C05104=1100.951,434.101,399.471,179.920,21.270,152.698
C05105=1100.945,433.854,399.513,179.918,21.260,152.696
C05106=1100.939,433.608,399.554,179.916,21.249,152.693
C05107=1100.933,433.362,399.596,179.915,21.239,152.691
C05108=1100.927,433.115,399.638,179.912,21.228,152.688
C05109=1100.921,432.869,399.679,179.911,21.218,152.686
C05110=1100.915,432.622,399.721,179.908,21.208,152.684
C05111=1100.909,432.376,399.762,179.907,21.197,152.682
C05112=1100.903,432.129,399.803,179.904,21.187,152.679
C05113=1100.897,431.883,399.844,179.903,21.177,152.677
C05114=1100.891,431.637,399.886,179.900,21.166,152.675
C05115=1100.886,431.391,399.927,179.899,21.157,152.673
C05116=1100.879,431.144,399.969,179.896,21.146,152.670
C05117=1100.873,430.897,400.010,179.894,21.136,152.668
C05118=1100.867,430.651,400.051,179.893,21.126,152.666
C05119=1100.861,430.405,400.093,179.890,21.116,152.664
C05120=1100.856,430.158,400.133,179.889,21.106,152.662
C05121=1100.850,429.912,400.175,179.886,21.096,152.659
C05122=1100.844,429.665,400.216,179.884,21.086,152.657
C05123=1100.838,429.419,400.257,179.883,21.076,152.655
C05124=1100.832,429.172,400.298,179.880,21.066,152.653
C05125=1100.827,428.926,400.339,179.878,21.057,152.651
C05126=1100.821,428.679,400.381,179.876,21.047,152.649
C05127=1100.815,428.433,400.421,179.874,21.037,152.647
C05128=1100.808,428.187,400.462,179.872,21.028,152.645
C05129=1100.803,427.940,400.503,179.870,21.018,152.643
C05130=1100.797,427.694,400.544,179.868,21.008,152.640
C05131=1100.791,427.447,400.585,179.866,20.999,152.638
C05132=1100.785,427.201,400.627,179.864,20.990,152.636
C05133=1100.779,426.954,400.667,179.862,20.980,152.634
C05134=1100.773,426.707,400.708,179.859,20.970,152.632
C05135=1100.767,426.461,400.749,179.857,20.961,152.630
C05136=1100.762,426.214,400.790,179.856,20.952,152.628
C05137=1100.755,425.968,400.830,179.854,20.942,152.626
C05138=1100.750,425.721,400.871,179.851,20.933,152.624
C05139=1100.744,425.475,400.912,179.849,20.924,152.622
C05140=1100.738,425.228,400.953,179.847,20.914,152.620
C05141=1100.733,425.005,400.989,179.845,20.906,152.619
C05142=1100.727,424.783,401.026,179.843,20.898,152.617
C05143=1100.722,424.561,401.063,179.841,20.889,152.615
C05144=1100.716,424.338,401.099,179.840,20.881,152.613
C05145=1100.711,424.115,401.136,179.837,20.873,152.611
C05146=1100.706,423.892,401.173,179.835,20.864,152.610
C05147=1100.701,423.670,401.210,179.833,20.857,152.608
C05148=1100.695,423.448,401.246,179.831,20.848,152.606
C05149=1100.690,423.202,401.286,179.829,20.839,152.604
C05150=1100.684,422.955,401.327,179.827,20.830,152.602
C05151=1100.678,422.708,401.367,179.825,20.821,152.601
C05152=1100.672,422.462,401.408,179.823,20.812,152.599
C05153=1100.666,422.215,401.448,179.821,20.804,152.597
C05154=1100.660,421.969,401.488,179.818,20.794,152.595
C05155=1100.654,421.722,401.529,179.816,20.786,152.593
C05156=1100.648,421.475,401.569,179.814,20.777,152.591
C05157=1100.643,421.229,401.610,179.812,20.768,152.590
C05158=1100.637,420.982,401.649,179.809,20.759,152.588
C05159=1100.631,420.735,401.690,179.807,20.751,152.586
C05160=1100.625,420.489,401.730,179.805,20.742,152.584
C05161=1100.618,420.242,401.770,179.803,20.733,152.582
C05162=1100.613,419.995,401.811,179.801,20.725,152.581
C05163=1100.607,419.749,401.850,179.798,20.716,152.579
C05164=1100.602,419.502,401.891,179.796,20.708,152.577
C05165=1100.595,419.256,401.931,179.794,20.699,152.575
C05166=1100.590,419.009,401.972,179.792,20.691,152.573
C05167=1100.584,418.762,402.011,179.790,20.682,152.572
C05168=1100.578,418.516,402.051,179.787,20.673,152.570
C05169=1100.572,418.269,402.092,179.785,20.665,152.568
C05170=1100.566,418.022,402.131,179.783,20.657,152.567
C05171=1100.560,417.775,402.172,179.780,20.649,152.565
C05172=1100.555,417.529,402.211,179.778,20.640,152.563
C05173=1100.549,417.282,402.251,179.776,20.632,152.561
C05174=1100.543,417.035,402.291,179.774,20.623,152.560
C05175=1100.537,416.788,402.331,179.771,20.615,152.558
C05176=1100.531,416.542,402.371,179.769,20.607,152.556
C05177=1100.526,416.295,402.411,179.767,20.599,152.555
C05178=1100.520,416.048,402.450,179.765,20.591,152.553
C05179=1100.513,415.801,402.491,179.762,20.583,152.552
C05180=1100.508,415.555,402.530,179.760,20.575,152.550
C05181=1100.501,415.308,402.570,179.758,20.566,152.548
C05182=1100.495,415.061,402.609,179.755,20.558,152.547
C05183=1100.491,414.814,402.649,179.753,20.551,152.545
C05184=1100.484,414.568,402.689,179.751,20.542,152.543
C05185=1100.478,414.321,402.728,179.748,20.534,152.542
C05186=1100.472,414.074,402.768,179.746,20.527,152.540
C05187=1100.466,413.828,402.808,179.744,20.519,152.539
C05188=1100.460,413.581,402.847,179.742,20.511,152.537
C05189=1100.454,413.333,402.887,179.739,20.503,152.535
C05190=1100.449,413.087,402.926,179.736,20.495,152.534
C05191=1100.442,412.840,402.966,179.735,20.487,152.532
C05192=1100.436,412.593,403.005,179.732,20.480,152.531
C05193=1100.431,412.347,403.045,179.730,20.472,152.529
C05194=1100.425,412.099,403.084,179.727,20.464,152.528
C05195=1100.420,411.853,403.123,179.725,20.457,152.526
C05196=1100.414,411.606,403.163,179.723,20.449,152.525
C05197=1100.409,411.390,403.197,179.721,20.442,152.524
C05198=1100.403,411.175,403.231,179.719,20.435,152.522
C05199=1100.398,410.960,403.266,179.717,20.429,152.521
C05200=1100.393,410.743,403.301,179.715,20.422,152.520
C05201=1100.388,410.528,403.335,179.713,20.416,152.518
C05202=1100.383,410.312,403.369,179.711,20.409,152.517
C05203=1100.378,410.097,403.403,179.709,20.402,152.516
C05204=1100.373,409.881,403.438,179.706,20.396,152.514
C05205=1100.367,409.634,403.477,179.704,20.388,152.513
C05206=1100.361,409.387,403.516,179.701,20.381,152.512
C05207=1100.355,409.140,403.556,179.699,20.373,152.510
C05208=1100.350,408.894,403.595,179.697,20.366,152.509
C05209=1100.344,408.646,403.633,179.695,20.359,152.507
C05210=1100.339,408.400,403.673,179.692,20.351,152.506
C05211=1100.333,408.153,403.712,179.689,20.344,152.504
C05212=1100.327,407.906,403.751,179.688,20.337,152.503
C05213=1100.320,407.659,403.790,179.685,20.329,152.502
C05214=1100.315,407.413,403.829,179.682,20.322,152.500
C05215=1100.309,407.165,403.868,179.680,20.315,152.499
C05216=1100.304,406.919,403.907,179.678,20.307,152.497
C05217=1100.297,406.672,403.946,179.676,20.300,152.496
C05218=1100.292,406.425,403.985,179.673,20.293,152.495
C05219=1100.286,406.178,404.023,179.670,20.286,152.493
C05220=1100.280,405.931,404.062,179.668,20.279,152.492
C05221=1100.275,405.685,404.101,179.665,20.272,152.491
C05222=1100.269,405.437,404.140,179.664,20.265,152.489
C05223=1100.263,405.191,404.179,179.661,20.257,152.488
C05224=1100.257,404.943,404.217,179.659,20.251,152.487
C05225=1100.251,404.697,404.256,179.656,20.243,152.485
C05226=1100.245,404.450,404.296,179.654,20.237,152.484
C05227=1100.239,404.203,404.334,179.651,20.230,152.483
C05228=1100.233,403.956,404.373,179.649,20.223,152.481
C05229=1100.228,403.709,404.411,179.646,20.216,152.480
C05230=1100.222,403.463,404.450,179.644,20.209,152.479
C05231=1100.216,403.215,404.489,179.641,20.202,152.477
C05232=1100.210,402.969,404.527,179.639,20.196,152.476
C05233=1100.204,402.721,404.566,179.636,20.189,152.475
C05234=1100.199,402.474,404.604,179.634,20.182,152.474
C05235=1100.193,402.228,404.643,179.631,20.175,152.473
C05236=1100.187,401.980,404.681,179.629,20.168,152.471
C05237=1100.181,401.734,404.720,179.627,20.162,152.470
C05238=1100.175,401.486,404.759,179.624,20.155,152.469
C05239=1100.169,401.239,404.796,179.622,20.148,152.468
C05240=1100.164,400.993,404.835,179.619,20.141,152.466
C05241=1100.158,400.745,404.874,179.617,20.135,152.465
C05242=1100.152,400.498,404.912,179.615,20.129,152.464
C05243=1100.147,400.251,404.950,179.612,20.121,152.463
C05244=1100.141,400.005,404.989,179.609,20.115,152.462
C05245=1100.135,399.757,405.027,179.607,20.108,152.460
C05246=1100.129,399.511,405.065,179.604,20.102,152.459
C05247=1100.124,399.264,405.103,179.602,20.096,152.458
C05248=1100.117,399.016,405.142,179.599,20.089,152.457
C05249=1100.111,398.770,405.180,179.597,20.083,152.456
C05250=1100.106,398.523,405.218,179.595,20.076,152.454
C05251=1100.099,398.276,405.257,179.592,20.070,152.453
C05252=1100.094,398.029,405.295,179.589,20.063,152.452
C05253=1100.089,397.813,405.328,179.587,20.058,152.451
C05254=1100.084,397.598,405.361,179.585,20.053,152.450
C05255=1100.079,397.382,405.394,179.583,20.047,152.449
C05256=1100.074,397.166,405.428,179.580,20.041,152.448
C05257=1100.069,396.951,405.460,179.578,20.036,152.447
C05258=1100.064,396.735,405.494,179.576,20.030,152.446
C05259=1100.059,396.520,405.527,179.574,20.025,152.445
C05260=1100.053,396.304,405.560,179.572,20.019,152.444
C05261=1100.048,396.057,405.598,179.570,20.013,152.443
C05262=1100.042,395.810,405.636,179.566,20.006,152.442
C05263=1100.036,395.563,405.674,179.564,20.001,152.441
C05264=1100.031,395.316,405.712,179.562,19.994,152.440
C05265=1100.025,395.069,405.750,179.560,19.988,152.439
C05266=1100.019,394.822,405.788,179.556,19.982,152.438
C05267=1100.013,394.576,405.826,179.554,19.976,152.437
C05268=1100.007,394.329,405.863,179.551,19.970,152.436
C05269=1100.002,394.080,405.901,179.549,19.964,152.435
C05270=1099.996,393.834,405.939,179.546,19.957,152.434
C05271=1099.990,393.587,405.977,179.543,19.952,152.433
C05272=1099.984,393.340,406.015,179.541,19.945,152.432
C05273=1099.978,393.093,406.052,179.539,19.940,152.431
C05274=1099.972,392.846,406.090,179.535,19.933,152.430
C05275=1099.967,392.599,406.128,179.533,19.927,152.428
C05276=1099.961,392.352,406.166,179.531,19.921,152.427
C05277=1099.955,392.105,406.204,179.528,19.916,152.426
C05278=1099.949,391.857,406.241,179.526,19.910,152.425
C05279=1099.943,391.611,406.279,179.522,19.904,152.425
C05280=1099.937,391.364,406.316,179.520,19.898,152.424
C05281=1099.932,391.117,406.353,179.518,19.892,152.423
C05282=1099.926,390.870,406.391,179.515,19.886,152.422
C05283=1099.920,390.622,406.428,179.513,19.881,152.421
C05284=1099.914,390.376,406.466,179.510,19.875,152.420
C05285=1099.909,390.129,406.504,179.507,19.869,152.419
C05286=1099.903,389.882,406.541,179.504,19.863,152.418
C05287=1099.896,389.635,406.578,179.502,19.857,152.417
C05288=1099.891,389.388,406.615,179.499,19.852,152.416
C05289=1099.885,389.141,406.653,179.497,19.846,152.415
C05290=1099.879,388.894,406.690,179.494,19.840,152.414
C05291=1099.873,388.647,406.727,179.491,19.835,152.413
C05292=1099.868,388.400,406.764,179.488,19.829,152.412
C05293=1099.862,388.153,406.802,179.485,19.823,152.411
C05294=1099.856,387.906,406.839,179.483,19.818,152.410
C05295=1099.851,387.658,406.876,179.480,19.812,152.409
C05296=1099.845,387.411,406.914,179.478,19.806,152.408
C05297=1099.838,387.164,406.950,179.475,19.801,152.408
C05298=1099.832,386.918,406.988,179.473,19.795,152.407
C05299=1099.827,386.670,407.025,179.470,19.790,152.406
C05300=1099.821,386.423,407.062,179.466,19.784,152.405
C05301=1099.815,386.176,407.100,179.464,19.778,152.404
C05302=1099.810,385.929,407.137,179.461,19.773,152.403
C05303=1099.803,385.682,407.174,179.459,19.768,152.402
C05304=1099.798,385.434,407.211,179.456,19.762,152.401
C05305=1099.792,385.188,407.248,179.453,19.757,152.401
C05306=1099.787,384.941,407.285,179.451,19.751,152.400
C05307=1099.781,384.694,407.322,179.448,19.746,152.399
C05308=1099.775,384.447,407.359,179.445,19.740,152.398
C05309=1099.770,384.237,407.391,179.443,19.736,152.397
C05310=1099.766,384.027,407.422,179.440,19.731,152.397
C05311=1099.761,383.819,407.453,179.438,19.727,152.396
C05312=1099.756,383.609,407.484,179.436,19.722,152.395
C05313=1099.751,383.400,407.516,179.433,19.717,152.394
C05314=1099.746,383.191,407.546,179.431,19.713,152.394
C05315=1099.736,382.772,407.609,179.427,19.704,152.392
C05316=1099.731,382.524,407.646,179.424,19.699,152.392
C05317=1099.725,382.277,407.683,179.422,19.693,152.391
C05318=1099.719,382.030,407.719,179.419,19.689,152.390
C05319=1099.714,381.783,407.756,179.416,19.683,152.389
C05320=1099.707,381.536,407.792,179.414,19.678,152.388
C05321=1099.702,381.289,407.829,179.411,19.673,152.388
C05322=1099.696,381.042,407.866,179.408,19.667,152.387
C05323=1099.690,380.794,407.903,179.405,19.663,152.386
C05324=1099.684,380.547,407.940,179.402,19.657,152.385
C05325=1099.678,380.300,407.976,179.399,19.652,152.385
C05326=1099.673,380.053,408.013,179.397,19.647,152.384
C05327=1099.667,379.806,408.050,179.394,19.642,152.383
C05328=1099.661,379.558,408.086,179.391,19.637,152.382
C05329=1099.655,379.311,408.122,179.388,19.632,152.381
C05330=1099.649,379.064,408.159,179.385,19.627,152.381
C05331=1099.644,378.818,408.195,179.383,19.622,152.380
C05332=1099.638,378.570,408.232,179.380,19.616,152.379
C05333=1099.632,378.323,408.268,179.377,19.611,152.379
C05334=1099.626,378.075,408.305,179.374,19.606,152.378
C05335=1099.621,377.829,408.341,179.371,19.601,152.377
C05336=1099.615,377.581,408.378,179.369,19.596,152.376
C05337=1099.609,377.334,408.414,179.366,19.591,152.376
C05338=1099.603,377.086,408.451,179.363,19.586,152.375
C05339=1099.598,376.840,408.487,179.361,19.582,152.374
C05340=1099.592,376.592,408.523,179.358,19.577,152.374
C05341=1099.586,376.345,408.560,179.355,19.572,152.373
C05342=1099.581,376.098,408.595,179.352,19.567,152.372
C05343=1099.575,375.851,408.632,179.349,19.562,152.371
C05344=1099.569,375.604,408.669,179.346,19.557,152.371
C05345=1099.564,375.356,408.705,179.343,19.552,152.370
C05346=1099.558,375.109,408.741,179.340,19.547,152.369
C05347=1099.552,374.862,408.777,179.338,19.542,152.369
C05348=1099.547,374.615,408.814,179.335,19.537,152.368
C05349=1099.541,374.367,408.849,179.333,19.533,152.367
C05350=1099.534,374.120,408.886,179.329,19.528,152.367
C05351=1099.530,373.873,408.922,179.327,19.523,152.366
C05352=1099.524,373.625,408.957,179.324,19.518,152.365
C05353=1099.517,373.378,408.994,179.321,19.514,152.365
C05354=1099.511,373.131,409.030,179.318,19.509,152.364
C05355=1099.505,372.884,409.066,179.315,19.504,152.364
C05356=1099.500,372.636,409.102,179.312,19.500,152.363
C05357=1099.494,372.389,409.138,179.309,19.495,152.362
C05358=1099.488,372.142,409.174,179.306,19.490,152.362
C05359=1099.482,371.895,409.210,179.303,19.486,152.361
C05360=1099.476,371.647,409.245,179.300,19.481,152.360
C05361=1099.471,371.400,409.281,179.298,19.477,152.360
C05362=1099.465,371.152,409.318,179.295,19.472,152.359
C05363=1099.460,370.906,409.353,179.292,19.467,152.359
C05364=1099.450,370.514,409.410,179.287,19.460,152.358
C05365=1099.441,370.122,409.466,179.283,19.453,152.357
C05366=1099.433,369.731,409.523,179.278,19.445,152.356
C05367=1099.423,369.339,409.580,179.273,19.438,152.355
C05368=1099.417,369.092,409.616,179.271,19.434,152.354
C05369=1099.411,368.845,409.651,179.268,19.429,152.354
C05370=1099.406,368.597,409.687,179.265,19.425,152.353
C05371=1099.401,368.350,409.723,179.262,19.420,152.353
C05372=1099.395,368.102,409.758,179.260,19.416,152.352
C05373=1099.389,367.855,409.794,179.257,19.412,152.351
C05374=1099.383,367.608,409.829,179.253,19.407,152.351
C05375=1099.377,367.360,409.865,179.250,19.402,152.350
C05376=1099.372,367.113,409.901,179.248,19.398,152.350
C05377=1099.366,366.865,409.936,179.245,19.393,152.349
C05378=1099.360,366.618,409.972,179.242,19.389,152.349
C05379=1099.354,366.371,410.007,179.239,19.384,152.348
C05380=1099.349,366.124,410.043,179.236,19.380,152.347
C05381=1099.343,365.876,410.079,179.233,19.376,152.347
C05382=1099.337,365.629,410.114,179.230,19.372,152.347
C05383=1099.332,365.381,410.149,179.227,19.367,152.346
C05384=1099.326,365.134,410.184,179.225,19.363,152.345
C05385=1099.320,364.886,410.220,179.222,19.359,152.345
C05386=1099.315,364.639,410.255,179.218,19.354,152.344
C05387=1099.308,364.392,410.290,179.215,19.350,152.344
C05388=1099.303,364.144,410.325,179.213,19.346,152.343
C05389=1099.297,363.896,410.361,179.210,19.342,152.343
C05390=1099.291,363.649,410.396,179.206,19.337,152.342
C05391=1099.286,363.402,410.432,179.204,19.333,152.342
C05392=1099.280,363.154,410.467,179.201,19.329,152.341
C05393=1099.274,362.908,410.501,179.198,19.325,152.341
C05394=1099.268,362.660,410.537,179.195,19.321,152.341
C05395=1099.263,362.413,410.572,179.192,19.316,152.340
C05396=1099.257,362.165,410.607,179.189,19.312,152.340
C05397=1099.251,361.918,410.643,179.186,19.308,152.339
C05398=1099.245,361.670,410.677,179.183,19.304,152.339
C05399=1099.240,361.423,410.713,179.180,19.300,152.338
C05400=1099.234,361.176,410.748,179.177,19.295,152.338
C05401=1099.228,360.927,410.783,179.174,19.291,152.337
C05402=1099.222,360.681,410.818,179.171,19.287,152.337
C05403=1099.216,360.432,410.853,179.168,19.283,152.336
C05404=1099.211,360.185,410.888,179.165,19.279,152.336
C05405=1099.206,359.938,410.923,179.162,19.275,152.335
C05406=1099.199,359.690,410.958,179.159,19.271,152.335
C05407=1099.194,359.443,410.993,179.156,19.267,152.335
C05408=1099.187,359.196,411.028,179.153,19.263,152.334
C05409=1099.182,358.948,411.062,179.150,19.259,152.334
C05410=1099.177,358.701,411.098,179.147,19.255,152.333
C05411=1099.170,358.453,411.132,179.144,19.251,152.333
C05412=1099.165,358.205,411.167,179.141,19.247,152.332
C05413=1099.160,357.958,411.202,179.138,19.243,152.332
C05414=1099.153,357.710,411.237,179.135,19.239,152.332
C05415=1099.148,357.463,411.272,179.132,19.235,152.331
C05416=1099.139,357.086,411.325,179.128,19.229,152.331
C05417=1099.131,356.710,411.377,179.123,19.223,152.330
C05418=1099.121,356.333,411.430,179.118,19.218,152.329
C05419=1099.112,355.957,411.483,179.114,19.211,152.329
C05420=1099.107,355.709,411.517,179.111,19.207,152.328
C05421=1099.101,355.462,411.552,179.108,19.204,152.328
C05422=1099.096,355.215,411.587,179.105,19.200,152.328
C05423=1099.090,354.967,411.621,179.101,19.195,152.327
C05424=1099.084,354.719,411.656,179.099,19.192,152.327
C05425=1099.079,354.472,411.690,179.095,19.188,152.327
C05426=1099.073,354.223,411.725,179.093,19.185,152.326
C05427=1099.067,353.977,411.760,179.089,19.180,152.326
C05428=1099.062,353.729,411.794,179.087,19.177,152.325
C05429=1099.056,353.482,411.828,179.084,19.173,152.325
C05430=1099.050,353.234,411.863,179.080,19.169,152.325
C05431=1099.044,352.986,411.897,179.077,19.165,152.324
C05432=1099.038,352.739,411.931,179.074,19.161,152.324
C05433=1099.033,352.492,411.966,179.071,19.158,152.324
C05434=1099.027,352.244,412.000,179.068,19.154,152.323
C05435=1099.022,351.996,412.035,179.065,19.150,152.323
C05436=1099.016,351.749,412.069,179.062,19.147,152.323
C05437=1099.010,351.501,412.103,179.059,19.143,152.322
C05438=1099.004,351.253,412.138,179.056,19.139,152.322
C05439=1098.998,351.006,412.172,179.053,19.136,152.322
C05440=1098.992,350.758,412.206,179.050,19.132,152.321
C05441=1098.987,350.511,412.240,179.046,19.128,152.321
C05442=1098.982,350.263,412.274,179.044,19.125,152.321
C05443=1098.975,350.015,412.309,179.040,19.121,152.320
C05444=1098.969,349.768,412.343,179.037,19.117,152.320
C05445=1098.964,349.520,412.377,179.034,19.113,152.320
C05446=1098.958,349.273,412.411,179.031,19.110,152.319
C05447=1098.953,349.026,412.446,179.028,19.106,152.319
C05448=1098.947,348.778,412.479,179.025,19.103,152.319
C05449=1098.941,348.529,412.514,179.022,19.099,152.318
C05450=1098.935,348.282,412.548,179.019,19.095,152.318
C05451=1098.930,348.035,412.582,179.016,19.092,152.318
C05452=1098.924,347.787,412.615,179.013,19.089,152.318
